LIN {X 0,Y 397.107,Z 581.021,A -85,B 0,C 180,E1 -11285.734,E2 -11285.734} C_VEL
LIN {X 0,Y 397.113,Z 581.016,A -85,B 0,C 180,E1 -11289.576,E2 -11289.576} C_VEL
LIN {X 0,Y 397.111,Z 581.016,A -85,B 0,C 180,E1 -11292.26,E2 -11292.26} C_VEL
LIN {X 0,Y 397.161,Z 581.009,A -85,B 0,C 180,E1 -11296.36,E2 -11296.36} C_VEL
LIN {X 0,Y 397.119,Z 581.014,A -85,B 0,C 180,E1 -11299.55,E2 -11299.55} C_VEL
LIN {X 0,Y 397.094,Z 581.019,A -85,B 0,C 180,E1 -11302.789,E2 -11302.789} C_VEL
LIN {X 0,Y 397.113,Z 581.011,A -85,B 0,C 180,E1 -11306.281,E2 -11306.281} C_VEL
LIN {X 0,Y 397.08,Z 581.018,A -85,B 0,C 180,E1 -11309.118,E2 -11309.118} C_VEL
LIN {X 0,Y 397.188,Z 581.007,A -85,B 0,C 180,E1 -11312.609,E2 -11312.609} C_VEL
LIN {X 0,Y 397.125,Z 581.014,A -85,B 0,C 180,E1 -11315.981,E2 -11315.981} C_VEL
LIN {X 0,Y 397.131,Z 581.012,A -85,B 0,C 180,E1 -11319.704,E2 -11319.704} C_VEL
LIN {X 0,Y 397.173,Z 581,A -85,B 0,C 180,E1 -11322.844,E2 -11322.844} C_VEL
LIN {X 0,Y 397.22,Z 581.007,A -85,B 0,C 180,E1 -11326.702,E2 -11326.702} C_VEL
LIN {X 0,Y 397.21,Z 580.998,A -85,B 0,C 180,E1 -11329.809,E2 -11329.809} C_VEL
LIN {X 0,Y 397.343,Z 580.986,A -85,B 0,C 180,E1 -11332.888,E2 -11332.888} C_VEL
LIN {X 0,Y 397.254,Z 581.001,A -85,B 0,C 180,E1 -11334.925,E2 -11334.925} C_VEL
LIN {X 0,Y 397.443,Z 580.964,A -85,B 0,C 180,E1 -11337.973,E2 -11337.973} C_VEL
LIN {X 0,Y 397.573,Z 580.952,A -85,B 0,C 180,E1 -11340,E2 -11340} C_VEL
LIN {X 0,Y 397.374,Z 580.984,A -85,B 0,C 180,E1 -11343.041,E2 -11343.041} C_VEL
LIN {X 0,Y 397.339,Z 580.977,A -85,B 0,C 180,E1 -11346.622,E2 -11346.622} C_VEL
LIN {X 0,Y 397.244,Z 581.002,A -85,B 0,C 180,E1 -11349.162,E2 -11349.162} C_VEL
LIN {X 0,Y 397.211,Z 580.994,A -85,B 0,C 180,E1 -11352.258,E2 -11352.258} C_VEL
LIN {X 0,Y 397.17,Z 581.011,A -85,B 0,C 180,E1 -11355.392,E2 -11355.392} C_VEL
LIN {X 0,Y 397.153,Z 581.004,A -85,B 0,C 180,E1 -11358.574,E2 -11358.574} C_VEL
LIN {X 0,Y 397.087,Z 581.019,A -85,B 0,C 180,E1 -11361.819,E2 -11361.819} C_VEL
LIN {X 0,Y 397.145,Z 581.011,A -85,B 0,C 180,E1 -11365.513,E2 -11365.513} C_VEL
LIN {X 0,Y 397.12,Z 581.016,A -85,B 0,C 180,E1 -11368.544,E2 -11368.544} C_VEL
LIN {X 0,Y 397.106,Z 581.017,A -85,B 0,C 180,E1 -11372.069,E2 -11372.069} C_VEL
LIN {X 0,Y 397.114,Z 581.019,A -85,B 0,C 180,E1 -11375.504,E2 -11375.504} C_VEL
LIN {X 0,Y 397.13,Z 581.017,A -85,B 0,C 180,E1 -11378.863,E2 -11378.863} C_VEL
LIN {X 0,Y 397.111,Z 580.995,A -85,B 0,C 180,E1 -11382.262,E2 -11382.262} C_VEL
LIN {X 0,Y 397.085,Z 581.023,A -85,B 0,C 180,E1 -11385.069,E2 -11385.069} C_VEL
LIN {X 0,Y 397.062,Z 581.012,A -85,B 0,C 180,E1 -11388.022,E2 -11388.022} C_VEL
LIN {X 0,Y 397.129,Z 581.012,A -85,B 0,C 180,E1 -11391.139,E2 -11391.139} C_VEL
LIN {X 0,Y 397.118,Z 581.016,A -85,B 0,C 180,E1 -11394.497,E2 -11394.497} C_VEL
LIN {X 0,Y 397.104,Z 581.02,A -85,B 0,C 180,E1 -11397.531,E2 -11397.531} C_VEL
LIN {X 0,Y 398.153,Z 583.972,A -85,B 0,C 180,E1 -11397.677,E2 -11397.677} C_VEL
LIN {X 0,Y 404.838,Z 599.166,A -85,B 0,C 180,E1 -11398.379,E2 -11398.379} C_VEL
LIN {X 0,Y 403.608,Z 681.671,A -85,B 0,C 180,E1 -11399.888,E2 -11399.888} C_VEL
LIN {X 0,Y 403.342,Z 694.362,A -85,B 0,C 180,E1 -11400.305,E2 -11400.305} C_VEL
LIN {X 0,Y 402.939,Z 705.504,A -85,B 0,C 180,E1 -11400.844,E2 -11400.844} C_VEL
LIN {X 0,Y 402.29,Z 716.836,A -85,B 0,C 180,E1 -11401.573,E2 -11401.573} C_VEL
LIN {X 0,Y 401.469,Z 728.036,A -85,B 0,C 180,E1 -11402.503,E2 -11402.503} C_VEL
LIN {X 0,Y 400.575,Z 738.584,A -85,B 0,C 180,E1 -11403.604,E2 -11403.604} C_VEL
LIN {X 0,Y 399.779,Z 747.58,A -85,B 0,C 180,E1 -11404.767,E2 -11404.767} C_VEL
LIN {X 0,Y 398.991,Z 755.975,A -85,B 0,C 180,E1 -11406.101,E2 -11406.101} C_VEL
LIN {X 0,Y 398.143,Z 764.097,A -85,B 0,C 180,E1 -11407.697,E2 -11407.697} C_VEL
LIN {X 0,Y 397.527,Z 770.543,A -85,B 0,C 180,E1 -11409.294,E2 -11409.294} C_VEL
LIN {X 0,Y 397.01,Z 775.554,A -85,B 0,C 180,E1 -11410.884,E2 -11410.884} C_VEL
LIN {X 0,Y 396.638,Z 779.358,A -85,B 0,C 180,E1 -11412.469,E2 -11412.469} C_VEL
LIN {X 0,Y 396.452,Z 781.287,A -85,B 0,C 180,E1 -11413.523,E2 -11413.523} C_VEL
LIN {X 0,Y 396.255,Z 782.789,A -85,B 0,C 180,E1 -11414.572,E2 -11414.572} C_VEL
LIN {X 0,Y 396.14,Z 783.814,A -85,B 0,C 180,E1 -11415.619,E2 -11415.619} C_VEL
LIN {X 0,Y 396.103,Z 784.664,A -85,B 0,C 180,E1 -11417.707,E2 -11417.707} C_VEL
LIN {X 0,Y 396.063,Z 784.463,A -85,B 0,C 180,E1 -11418.744,E2 -11418.744} C_VEL
LIN {X 0,Y 396.135,Z 782.858,A -85,B 0,C 180,E1 -11420.812,E2 -11420.812} C_VEL
LIN {X 0,Y 396.234,Z 781.448,A -85,B 0,C 180,E1 -11421.843,E2 -11421.843} C_VEL
LIN {X 0,Y 396.459,Z 779.154,A -85,B 0,C 180,E1 -11423.078,E2 -11423.078} C_VEL
LIN {X 0,Y 396.744,Z 774.546,A -85,B 0,C 180,E1 -11424.919,E2 -11424.919} C_VEL
LIN {X 0,Y 397.06,Z 769.443,A -85,B 0,C 180,E1 -11426.448,E2 -11426.448} C_VEL
LIN {X 0,Y 397.584,Z 763.023,A -85,B 0,C 180,E1 -11427.974,E2 -11427.974} C_VEL
LIN {X 0,Y 398.172,Z 755.074,A -85,B 0,C 180,E1 -11429.494,E2 -11429.494} C_VEL
LIN {X 0,Y 398.92,Z 746.903,A -85,B 0,C 180,E1 -11430.757,E2 -11430.757} C_VEL
LIN {X 0,Y 399.601,Z 736.901,A -85,B 0,C 180,E1 -11432.016,E2 -11432.016} C_VEL
LIN {X 0,Y 400.368,Z 725.703,A -85,B 0,C 180,E1 -11433.145,E2 -11433.145} C_VEL
LIN {X 0,Y 400.855,Z 718.327,A -85,B 0,C 180,E1 -11433.746,E2 -11433.746} C_VEL
LIN {X 0,Y 400.522,Z 713.137,A -85,B 0,C 180,E1 -11434.145,E2 -11434.145} C_VEL
LIN {X 0,Y 398.165,Z 704.558,A -85,B 0,C 180,E1 -11434.779,E2 -11434.779} C_VEL
LIN {X 0,Y 395.699,Z 695.737,A -85,B 0,C 180,E1 -11435.325,E2 -11435.325} C_VEL
LIN {X 0,Y 395.17,Z 690.125,A -85,B 0,C 180,E1 -11435.573,E2 -11435.573} C_VEL
LIN {X 0,Y 395.439,Z 677.057,A -85,B 0,C 180,E1 -11435.929,E2 -11435.929} C_VEL
LIN {X 0,Y 396.414,Z 599.082,A -85,B 0,C 180,E1 -11437.34,E2 -11437.34} C_VEL
LIN {X 0,Y 390.306,Z 581.87,A -85,B 0,C 180,E1 -11437.965,E2 -11437.965} C_VEL
LIN {X 0,Y 390.16,Z 581.883,A -85,B 0,C 180,E1 -11441.428,E2 -11441.428} C_VEL
LIN {X 0,Y 390.149,Z 581.885,A -85,B 0,C 180,E1 -11444.607,E2 -11444.607} C_VEL
LIN {X 0,Y 390.129,Z 581.891,A -85,B 0,C 180,E1 -11447.833,E2 -11447.833} C_VEL
LIN {X 0,Y 390.056,Z 581.893,A -85,B 0,C 180,E1 -11451.122,E2 -11451.122} C_VEL
LIN {X 0,Y 390.073,Z 581.895,A -85,B 0,C 180,E1 -11454.48,E2 -11454.48} C_VEL
LIN {X 0,Y 390.107,Z 581.919,A -85,B 0,C 180,E1 -11455.872,E2 -11455.872} C_VEL
LIN {X 0,Y 396.737,Z 599.495,A -85,B 0,C 180,E1 -11456.558,E2 -11456.558} C_VEL
LIN {X 0,Y 395.49,Z 682.574,A -85,B 0,C 180,E1 -11458.183,E2 -11458.183} C_VEL
LIN {X 0,Y 395.145,Z 696.043,A -85,B 0,C 180,E1 -11458.663,E2 -11458.663} C_VEL
LIN {X 0,Y 394.709,Z 707.466,A -85,B 0,C 180,E1 -11459.253,E2 -11459.253} C_VEL
LIN {X 0,Y 394.113,Z 718.824,A -85,B 0,C 180,E1 -11460.027,E2 -11460.027} C_VEL
LIN {X 0,Y 393.39,Z 730.372,A -85,B 0,C 180,E1 -11461.046,E2 -11461.046} C_VEL
LIN {X 0,Y 392.604,Z 740.657,A -85,B 0,C 180,E1 -11462.177,E2 -11462.177} C_VEL
LIN {X 0,Y 391.83,Z 750.29,A -85,B 0,C 180,E1 -11463.487,E2 -11463.487} C_VEL
LIN {X 0,Y 391.14,Z 758.584,A -85,B 0,C 180,E1 -11464.884,E2 -11464.884} C_VEL
LIN {X 0,Y 390.469,Z 766.071,A -85,B 0,C 180,E1 -11466.438,E2 -11466.438} C_VEL
LIN {X 0,Y 390.018,Z 772.477,A -85,B 0,C 180,E1 -11468.109,E2 -11468.109} C_VEL
LIN {X 0,Y 389.575,Z 777.532,A -85,B 0,C 180,E1 -11469.822,E2 -11469.822} C_VEL
LIN {X 0,Y 389.315,Z 780.786,A -85,B 0,C 180,E1 -11471.272,E2 -11471.272} C_VEL
LIN {X 0,Y 389.164,Z 782.437,A -85,B 0,C 180,E1 -11472.232,E2 -11472.232} C_VEL
LIN {X 0,Y 389.023,Z 784.323,A -85,B 0,C 180,E1 -11473.728,E2 -11473.728} C_VEL
LIN {X 0,Y 388.955,Z 785.325,A -85,B 0,C 180,E1 -11475.195,E2 -11475.195} C_VEL
LIN {X 0,Y 388.95,Z 785.526,A -85,B 0,C 180,E1 -11476.636,E2 -11476.636} C_VEL
LIN {X 0,Y 389.025,Z 784.989,A -85,B 0,C 180,E1 -11478.054,E2 -11478.054} C_VEL
LIN {X 0,Y 389.185,Z 783.734,A -85,B 0,C 180,E1 -11479.451,E2 -11479.451} C_VEL
LIN {X 0,Y 389.545,Z 780.384,A -85,B 0,C 180,E1 -11481.54,E2 -11481.54} C_VEL
LIN {X 0,Y 389.864,Z 776.967,A -85,B 0,C 180,E1 -11483.005,E2 -11483.005} C_VEL
LIN {X 0,Y 390.382,Z 771.36,A -85,B 0,C 180,E1 -11484.824,E2 -11484.824} C_VEL
LIN {X 0,Y 391.044,Z 764.821,A -85,B 0,C 180,E1 -11486.451,E2 -11486.451} C_VEL
LIN {X 0,Y 391.877,Z 756.375,A -85,B 0,C 180,E1 -11488.106,E2 -11488.106} C_VEL
LIN {X 0,Y 392.628,Z 748.547,A -85,B 0,C 180,E1 -11489.349,E2 -11489.349} C_VEL
LIN {X 0,Y 393.456,Z 739.523,A -85,B 0,C 180,E1 -11490.529,E2 -11490.529} C_VEL
LIN {X 0,Y 394.26,Z 728.785,A -85,B 0,C 180,E1 -11491.666,E2 -11491.666} C_VEL
LIN {X 0,Y 395.106,Z 716.39,A -85,B 0,C 180,E1 -11492.689,E2 -11492.689} C_VEL
LIN {X 0,Y 395.759,Z 704.167,A -85,B 0,C 180,E1 -11493.452,E2 -11493.452} C_VEL
LIN {X 0,Y 396.157,Z 690.604,A -85,B 0,C 180,E1 -11494.055,E2 -11494.055} C_VEL
LIN {X 0,Y 396.419,Z 678.086,A -85,B 0,C 180,E1 -11494.404,E2 -11494.404} C_VEL
LIN {X 0,Y 397.8,Z 600.33,A -85,B 0,C 180,E1 -11495.932,E2 -11495.932} C_VEL
LIN {X 0,Y 390.166,Z 582.414,A -85,B 0,C 180,E1 -11496.794,E2 -11496.794} C_VEL
LIN {X 0,Y 390.076,Z 581.896,A -85,B 0,C 180,E1 -11496.817,E2 -11496.817} C_VEL
LIN {X 0,Y 390.096,Z 581.894,A -85,B 0,C 180,E1 -11499.983,E2 -11499.983} C_VEL
LIN {X 0,Y 390.13,Z 581.889,A -85,B 0,C 180,E1 -11503.248,E2 -11503.248} C_VEL
LIN {X 0,Y 390.186,Z 581.883,A -85,B 0,C 180,E1 -11506.561,E2 -11506.561} C_VEL
LIN {X 0,Y 390.171,Z 581.883,A -85,B 0,C 180,E1 -11509.623,E2 -11509.623} C_VEL
LIN {X 0,Y 390.31,Z 581.866,A -85,B 0,C 180,E1 -11512.759,E2 -11512.759} C_VEL
LIN {X 0,Y 390.225,Z 581.875,A -85,B 0,C 180,E1 -11514.833,E2 -11514.833} C_VEL
LIN {X 0,Y 390.412,Z 581.849,A -85,B 0,C 180,E1 -11517.937,E2 -11517.937} C_VEL
LIN {X 0,Y 390.543,Z 581.837,A -85,B 0,C 180,E1 -11520,E2 -11520} C_VEL
LIN {X 0,Y 390.308,Z 581.861,A -85,B 0,C 180,E1 -11523.097,E2 -11523.097} C_VEL
LIN {X 0,Y 390.33,Z 581.863,A -85,B 0,C 180,E1 -11526.202,E2 -11526.202} C_VEL
LIN {X 0,Y 390.201,Z 581.873,A -85,B 0,C 180,E1 -11529.329,E2 -11529.329} C_VEL
LIN {X 0,Y 390.169,Z 581.88,A -85,B 0,C 180,E1 -11532.483,E2 -11532.483} C_VEL
LIN {X 0,Y 390.131,Z 581.882,A -85,B 0,C 180,E1 -11535.677,E2 -11535.677} C_VEL
LIN {X 0,Y 390.097,Z 581.888,A -85,B 0,C 180,E1 -11538.923,E2 -11538.923} C_VEL
LIN {X 0,Y 390.033,Z 581.899,A -85,B 0,C 180,E1 -11542.235,E2 -11542.235} C_VEL
LIN {X 0,Y 390.112,Z 581.889,A -85,B 0,C 180,E1 -11545.744,E2 -11545.744} C_VEL
LIN {X 0,Y 390.059,Z 581.896,A -85,B 0,C 180,E1 -11549.11,E2 -11549.11} C_VEL
LIN {X 0,Y 390.037,Z 581.899,A -85,B 0,C 180,E1 -11552.722,E2 -11552.722} C_VEL
LIN {X 0,Y 390.052,Z 581.897,A -85,B 0,C 180,E1 -11555.826,E2 -11555.826} C_VEL
LIN {X 0,Y 390.07,Z 581.893,A -85,B 0,C 180,E1 -11559.22,E2 -11559.22} C_VEL
LIN {X 0,Y 390.116,Z 581.891,A -85,B 0,C 180,E1 -11562.388,E2 -11562.388} C_VEL
LIN {X 0,Y 390.057,Z 581.897,A -85,B 0,C 180,E1 -11565.358,E2 -11565.358} C_VEL
LIN {X 0,Y 390.065,Z 581.898,A -85,B 0,C 180,E1 -11568.192,E2 -11568.192} C_VEL
LIN {X 0,Y 390.092,Z 581.894,A -85,B 0,C 180,E1 -11570.909,E2 -11570.909} C_VEL
LIN {X 0,Y 390.084,Z 581.894,A -85,B 0,C 180,E1 -11574.794,E2 -11574.794} C_VEL
LIN {X 0,Y 390.073,Z 582.026,A -85,B 0,C 180,E1 -11578.363,E2 -11578.363} C_VEL
LIN {X 0,Y 392.97,Z 594.47,A -85,B 0,C 180,E1 -11581.127,E2 -11581.127} C_VEL
LIN {X 0,Y 394.598,Z 603.068,A -85,B 0,C 180,E1 -11582.94,E2 -11582.94} C_VEL
LIN {X 0,Y 393.842,Z 613.598,A -85,B 0,C 180,E1 -11584.925,E2 -11584.925} C_VEL
LIN {X 0,Y 392.147,Z 635.612,A -85,B 0,C 180,E1 -11588.996,E2 -11588.996} C_VEL
LIN {X 0,Y 392.035,Z 636.9,A -85,B 0,C 180,E1 -11589.231,E2 -11589.231} C_VEL
LIN {X 0,Y 395.926,Z 664.717,A -85,B 0,C 180,E1 -11590.051,E2 -11590.051} C_VEL
LIN {X 0,Y 396.965,Z 675.261,A -85,B 0,C 180,E1 -11590.325,E2 -11590.325} C_VEL
LIN {X 0,Y 395.717,Z 747.647,A -85,B 0,C 180,E1 -11591.759,E2 -11591.759} C_VEL
LIN {X 0,Y 395.033,Z 761.284,A -85,B 0,C 180,E1 -11592.229,E2 -11592.229} C_VEL
LIN {X 0,Y 394.133,Z 774.25,A -85,B 0,C 180,E1 -11592.89,E2 -11592.89} C_VEL
LIN {X 0,Y 393.186,Z 786.925,A -85,B 0,C 180,E1 -11593.783,E2 -11593.783} C_VEL
LIN {X 0,Y 392.18,Z 798.275,A -85,B 0,C 180,E1 -11594.807,E2 -11594.807} C_VEL
LIN {X 0,Y 391.42,Z 808.805,A -85,B 0,C 180,E1 -11596.003,E2 -11596.003} C_VEL
LIN {X 0,Y 390.496,Z 817.885,A -85,B 0,C 180,E1 -11597.264,E2 -11597.264} C_VEL
LIN {X 0,Y 389.799,Z 827.014,A -85,B 0,C 180,E1 -11598.824,E2 -11598.824} C_VEL
LIN {X 0,Y 389.327,Z 834.372,A -85,B 0,C 180,E1 -11600.388,E2 -11600.388} C_VEL
LIN {X 0,Y 389.037,Z 841.107,A -85,B 0,C 180,E1 -11602.213,E2 -11602.213} C_VEL
LIN {X 0,Y 388.903,Z 845.58,A -85,B 0,C 180,E1 -11603.775,E2 -11603.775} C_VEL
LIN {X 0,Y 388.942,Z 847.974,A -85,B 0,C 180,E1 -11604.817,E2 -11604.817} C_VEL
LIN {X 0,Y 388.856,Z 849.875,A -85,B 0,C 180,E1 -11605.854,E2 -11605.854} C_VEL
LIN {X 0,Y 388.997,Z 851.337,A -85,B 0,C 180,E1 -11606.893,E2 -11606.893} C_VEL
LIN {X 0,Y 389.023,Z 852.379,A -85,B 0,C 180,E1 -11607.929,E2 -11607.929} C_VEL
LIN {X 0,Y 389.002,Z 853.016,A -85,B 0,C 180,E1 -11608.965,E2 -11608.965} C_VEL
LIN {X 0,Y 388.967,Z 853.206,A -85,B 0,C 180,E1 -11610,E2 -11610} C_VEL
LIN {X 0,Y 389.002,Z 852.98,A -85,B 0,C 180,E1 -11611.035,E2 -11611.035} C_VEL
LIN {X 0,Y 389.049,Z 852.354,A -85,B 0,C 180,E1 -11612.07,E2 -11612.07} C_VEL
LIN {X 0,Y 389,Z 851.311,A -85,B 0,C 180,E1 -11613.107,E2 -11613.107} C_VEL
LIN {X 0,Y 388.869,Z 849.793,A -85,B 0,C 180,E1 -11614.146,E2 -11614.146} C_VEL
LIN {X 0,Y 388.926,Z 846.715,A -85,B 0,C 180,E1 -11615.704,E2 -11615.704} C_VEL
LIN {X 0,Y 388.935,Z 842.53,A -85,B 0,C 180,E1 -11617.267,E2 -11617.267} C_VEL
LIN {X 0,Y 389.207,Z 836.12,A -85,B 0,C 180,E1 -11619.091,E2 -11619.091} C_VEL
LIN {X 0,Y 389.596,Z 829.127,A -85,B 0,C 180,E1 -11620.655,E2 -11620.655} C_VEL
LIN {X 0,Y 390.39,Z 819.171,A -85,B 0,C 180,E1 -11622.476,E2 -11622.476} C_VEL
LIN {X 0,Y 391.218,Z 809.61,A -85,B 0,C 180,E1 -11623.878,E2 -11623.878} C_VEL
LIN {X 0,Y 392.057,Z 799.634,A -85,B 0,C 180,E1 -11625.065,E2 -11625.065} C_VEL
LIN {X 0,Y 393.058,Z 788.861,A -85,B 0,C 180,E1 -11626.089,E2 -11626.089} C_VEL
LIN {X 0,Y 394.062,Z 776.778,A -85,B 0,C 180,E1 -11626.98,E2 -11626.98} C_VEL
LIN {X 0,Y 394.884,Z 764.155,A -85,B 0,C 180,E1 -11627.678,E2 -11627.678} C_VEL
LIN {X 0,Y 395.592,Z 751.57,A -85,B 0,C 180,E1 -11628.147,E2 -11628.147} C_VEL
LIN {X 0,Y 395.948,Z 735.695,A -85,B 0,C 180,E1 -11628.498,E2 -11628.498} C_VEL
LIN {X 0,Y 396.808,Z 671.548,A -85,B 0,C 180,E1 -11629.684,E2 -11629.684} C_VEL
LIN {X 0,Y 392.936,Z 639.109,A -85,B 0,C 180,E1 -11630.548,E2 -11630.548} C_VEL
LIN {X 0,Y 392.608,Z 636.373,A -85,B 0,C 180,E1 -11630.635,E2 -11630.635} C_VEL
LIN {X 0,Y 394.524,Z 610.695,A -85,B 0,C 180,E1 -11634.7,E2 -11634.7} C_VEL
LIN {X 0,Y 394.953,Z 603.562,A -85,B 0,C 180,E1 -11635.846,E2 -11635.846} C_VEL
LIN {X 0,Y 391.748,Z 588.885,A -85,B 0,C 180,E1 -11638.47,E2 -11638.47} C_VEL
LIN {X 0,Y 390.068,Z 581.896,A -85,B 0,C 180,E1 -11639.78,E2 -11639.78} C_VEL
LIN {X 0,Y 390.042,Z 581.899,A -85,B 0,C 180,E1 -11642.721,E2 -11642.721} C_VEL
LIN {X 0,Y 390.056,Z 581.901,A -85,B 0,C 180,E1 -11645.825,E2 -11645.825} C_VEL
LIN {X 0,Y 390.071,Z 581.892,A -85,B 0,C 180,E1 -11649.218,E2 -11649.218} C_VEL
LIN {X 0,Y 390.077,Z 581.892,A -85,B 0,C 180,E1 -11652.379,E2 -11652.379} C_VEL
LIN {X 0,Y 390.101,Z 581.887,A -85,B 0,C 180,E1 -11656.105,E2 -11656.105} C_VEL
LIN {X 0,Y 390.078,Z 581.89,A -85,B 0,C 180,E1 -11659.173,E2 -11659.173} C_VEL
LIN {X 0,Y 390.042,Z 581.901,A -85,B 0,C 180,E1 -11662.448,E2 -11662.448} C_VEL
LIN {X 0,Y 390.062,Z 581.887,A -85,B 0,C 180,E1 -11666.044,E2 -11666.044} C_VEL
LIN {X 0,Y 390.042,Z 581.9,A -85,B 0,C 180,E1 -11668.497,E2 -11668.497} C_VEL
LIN {X 0,Y 390.11,Z 581.88,A -85,B 0,C 180,E1 -11672.069,E2 -11672.069} C_VEL
LIN {X 0,Y 390.072,Z 581.891,A -85,B 0,C 180,E1 -11675.519,E2 -11675.519} C_VEL
LIN {X 0,Y 390.047,Z 581.896,A -85,B 0,C 180,E1 -11678.877,E2 -11678.877} C_VEL
LIN {X 0,Y 390.12,Z 581.889,A -85,B 0,C 180,E1 -11682.166,E2 -11682.166} C_VEL
LIN {X 0,Y 390.135,Z 581.879,A -85,B 0,C 180,E1 -11685.392,E2 -11685.392} C_VEL
LIN {X 0,Y 390.14,Z 581.886,A -85,B 0,C 180,E1 -11688.571,E2 -11688.571} C_VEL
LIN {X 0,Y 390.298,Z 581.852,A -85,B 0,C 180,E1 -11692.032,E2 -11692.032} C_VEL
LIN {X 0,Y 390.226,Z 581.878,A -85,B 0,C 180,E1 -11694.833,E2 -11694.833} C_VEL
LIN {X 0,Y 390.412,Z 581.839,A -85,B 0,C 180,E1 -11697.937,E2 -11697.937} C_VEL
LIN {X 0,Y 390.543,Z 581.827,A -85,B 0,C 180,E1 -11700,E2 -11700} C_VEL
LIN {X 0,Y 390.308,Z 581.863,A -85,B 0,C 180,E1 -11703.097,E2 -11703.097} C_VEL
LIN {X 0,Y 390.295,Z 581.854,A -85,B 0,C 180,E1 -11706.616,E2 -11706.616} C_VEL
LIN {X 0,Y 390.196,Z 581.879,A -85,B 0,C 180,E1 -11709.329,E2 -11709.329} C_VEL
LIN {X 0,Y 390.186,Z 581.875,A -85,B 0,C 180,E1 -11713.439,E2 -11713.439} C_VEL
LIN {X 0,Y 390.14,Z 581.881,A -85,B 0,C 180,E1 -11717.308,E2 -11717.308} C_VEL
LIN {X 0,Y 390.079,Z 581.888,A -85,B 0,C 180,E1 -11720.47,E2 -11720.47} C_VEL
LIN {X 0,Y 390.07,Z 581.887,A -85,B 0,C 180,E1 -11724.481,E2 -11724.481} C_VEL
LIN {X 0,Y 390.109,Z 581.888,A -85,B 0,C 180,E1 -11728.026,E2 -11728.026} C_VEL
LIN {X 0,Y 390.043,Z 581.9,A -85,B 0,C 180,E1 -11731.503,E2 -11731.503} C_VEL
LIN {X 0,Y 390.08,Z 581.891,A -85,B 0,C 180,E1 -11735.208,E2 -11735.208} C_VEL
LIN {X 0,Y 390.089,Z 581.897,A -85,B 0,C 180,E1 -11739.093,E2 -11739.093} C_VEL
LIN {X 0,Y 390.077,Z 581.87,A -85,B 0,C 180,E1 -11742.381,E2 -11742.381} C_VEL
LIN {X 0,Y 390.051,Z 581.894,A -85,B 0,C 180,E1 -11746.115,E2 -11746.115} C_VEL
LIN {X 0,Y 390.053,Z 581.899,A -85,B 0,C 180,E1 -11749.561,E2 -11749.561} C_VEL
LIN {X 0,Y 390.043,Z 581.89,A -85,B 0,C 180,E1 -11752.45,E2 -11752.45} C_VEL
LIN {X 0,Y 390.066,Z 581.896,A -85,B 0,C 180,E1 -11755.976,E2 -11755.976} C_VEL
LIN {X 0,Y 390.061,Z 581.897,A -85,B 0,C 180,E1 -11757.098,E2 -11757.098} C_VEL
LIN {X 0,Y 391.138,Z 584.861,A -85,B 0,C 180,E1 -11757.24,E2 -11757.24} C_VEL
LIN {X 0,Y 398.258,Z 600.928,A -85,B 0,C 180,E1 -11758.011,E2 -11758.011} C_VEL
LIN {X 0,Y 397.013,Z 682.018,A -85,B 0,C 180,E1 -11759.518,E2 -11759.518} C_VEL
LIN {X 0,Y 396.752,Z 694.64,A -85,B 0,C 180,E1 -11759.937,E2 -11759.937} C_VEL
LIN {X 0,Y 396.302,Z 705.838,A -85,B 0,C 180,E1 -11760.48,E2 -11760.48} C_VEL
LIN {X 0,Y 395.646,Z 717.052,A -85,B 0,C 180,E1 -11761.205,E2 -11761.205} C_VEL
LIN {X 0,Y 394.79,Z 728.228,A -85,B 0,C 180,E1 -11762.142,E2 -11762.142} C_VEL
LIN {X 0,Y 393.825,Z 739.065,A -85,B 0,C 180,E1 -11763.286,E2 -11763.286} C_VEL
LIN {X 0,Y 392.902,Z 748.814,A -85,B 0,C 180,E1 -11764.578,E2 -11764.578} C_VEL
LIN {X 0,Y 391.946,Z 758.19,A -85,B 0,C 180,E1 -11766.133,E2 -11766.133} C_VEL
LIN {X 0,Y 391.205,Z 765.125,A -85,B 0,C 180,E1 -11767.558,E2 -11767.558} C_VEL
LIN {X 0,Y 390.645,Z 770.502,A -85,B 0,C 180,E1 -11768.912,E2 -11768.912} C_VEL
LIN {X 0,Y 390.075,Z 775.688,A -85,B 0,C 180,E1 -11770.53,E2 -11770.53} C_VEL
LIN {X 0,Y 389.647,Z 779.619,A -85,B 0,C 180,E1 -11772.144,E2 -11772.144} C_VEL
LIN {X 0,Y 389.458,Z 781.604,A -85,B 0,C 180,E1 -11773.219,E2 -11773.219} C_VEL
LIN {X 0,Y 389.245,Z 783.166,A -85,B 0,C 180,E1 -11774.287,E2 -11774.287} C_VEL
LIN {X 0,Y 389.094,Z 784.294,A -85,B 0,C 180,E1 -11775.353,E2 -11775.353} C_VEL
LIN {X 0,Y 389.053,Z 785.244,A -85,B 0,C 180,E1 -11777.481,E2 -11777.481} C_VEL
LIN {X 0,Y 389.007,Z 785.138,A -85,B 0,C 180,E1 -11778.537,E2 -11778.537} C_VEL
LIN {X 0,Y 389.067,Z 783.643,A -85,B 0,C 180,E1 -11780.644,E2 -11780.644} C_VEL
LIN {X 0,Y 389.148,Z 782.309,A -85,B 0,C 180,E1 -11781.693,E2 -11781.693} C_VEL
LIN {X 0,Y 389.382,Z 779.851,A -85,B 0,C 180,E1 -11783.075,E2 -11783.075} C_VEL
LIN {X 0,Y 389.676,Z 775.632,A -85,B 0,C 180,E1 -11784.826,E2 -11784.826} C_VEL
LIN {X 0,Y 389.997,Z 770.674,A -85,B 0,C 180,E1 -11786.384,E2 -11786.384} C_VEL
LIN {X 0,Y 390.525,Z 764.398,A -85,B 0,C 180,E1 -11787.937,E2 -11787.937} C_VEL
LIN {X 0,Y 391.1,Z 756.611,A -85,B 0,C 180,E1 -11789.485,E2 -11789.485} C_VEL
LIN {X 0,Y 391.854,Z 748.635,A -85,B 0,C 180,E1 -11790.771,E2 -11790.771} C_VEL
LIN {X 0,Y 392.595,Z 738.95,A -85,B 0,C 180,E1 -11792.052,E2 -11792.052} C_VEL
LIN {X 0,Y 393.34,Z 728.066,A -85,B 0,C 180,E1 -11793.201,E2 -11793.201} C_VEL
LIN {X 0,Y 394.063,Z 717.452,A -85,B 0,C 180,E1 -11794.091,E2 -11794.091} C_VEL
LIN {X 0,Y 394.692,Z 704.664,A -85,B 0,C 180,E1 -11794.916,E2 -11794.916} C_VEL
LIN {X 0,Y 395.13,Z 691.574,A -85,B 0,C 180,E1 -11795.518,E2 -11795.518} C_VEL
LIN {X 0,Y 395.17,Z 690.125,A -85,B 0,C 180,E1 -11795.573,E2 -11795.573} C_VEL
LIN {X 0,Y 394.652,Z 684.425,A -85,B 0,C 180,E1 -11795.786,E2 -11795.786} C_VEL
LIN {X 0,Y 389.395,Z 665.772,A -85,B 0,C 180,E1 -11796.397,E2 -11796.397} C_VEL
LIN {X 0,Y 388.838,Z 659.957,A -85,B 0,C 180,E1 -11796.524,E2 -11796.524} C_VEL
LIN {X 0,Y 389.489,Z 600.174,A -85,B 0,C 180,E1 -11797.63,E2 -11797.63} C_VEL
LIN {X 0,Y 383.259,Z 582.747,A -85,B 0,C 180,E1 -11798.27,E2 -11798.27} C_VEL
LIN {X 0,Y 383.109,Z 582.763,A -85,B 0,C 180,E1 -11801.641,E2 -11801.641} C_VEL
LIN {X 0,Y 383.114,Z 582.76,A -85,B 0,C 180,E1 -11804.881,E2 -11804.881} C_VEL
LIN {X 0,Y 383.091,Z 582.768,A -85,B 0,C 180,E1 -11808.172,E2 -11808.172} C_VEL
LIN {X 0,Y 382.993,Z 582.775,A -85,B 0,C 180,E1 -11811.53,E2 -11811.53} C_VEL
LIN {X 0,Y 383.056,Z 582.768,A -85,B 0,C 180,E1 -11815.25,E2 -11815.25} C_VEL
LIN {X 0,Y 383.057,Z 582.769,A -85,B 0,C 180,E1 -11815.504,E2 -11815.504} C_VEL
LIN {X 0,Y 387.907,Z 595.517,A -85,B 0,C 180,E1 -11816.041,E2 -11816.041} C_VEL
LIN {X 0,Y 390.045,Z 601.164,A -85,B 0,C 180,E1 -11816.265,E2 -11816.265} C_VEL
LIN {X 0,Y 388.688,Z 683.075,A -85,B 0,C 180,E1 -11817.894,E2 -11817.894} C_VEL
LIN {X 0,Y 388.347,Z 696.518,A -85,B 0,C 180,E1 -11818.38,E2 -11818.38} C_VEL
LIN {X 0,Y 387.784,Z 709.508,A -85,B 0,C 180,E1 -11819.073,E2 -11819.073} C_VEL
LIN {X 0,Y 387.095,Z 721.91,A -85,B 0,C 180,E1 -11819.979,E2 -11819.979} C_VEL
LIN {X 0,Y 386.313,Z 733.533,A -85,B 0,C 180,E1 -11821.07,E2 -11821.07} C_VEL
LIN {X 0,Y 385.548,Z 743.292,A -85,B 0,C 180,E1 -11822.22,E2 -11822.22} C_VEL
LIN {X 0,Y 384.746,Z 752.441,A -85,B 0,C 180,E1 -11823.542,E2 -11823.542} C_VEL
LIN {X 0,Y 384.093,Z 760.013,A -85,B 0,C 180,E1 -11824.874,E2 -11824.874} C_VEL
LIN {X 0,Y 383.478,Z 766.506,A -85,B 0,C 180,E1 -11826.255,E2 -11826.255} C_VEL
LIN {X 0,Y 383.035,Z 772.783,A -85,B 0,C 180,E1 -11827.91,E2 -11827.91} C_VEL
LIN {X 0,Y 382.578,Z 777.551,A -85,B 0,C 180,E1 -11829.507,E2 -11829.507} C_VEL
LIN {X 0,Y 382.22,Z 781.806,A -85,B 0,C 180,E1 -11831.447,E2 -11831.447} C_VEL
LIN {X 0,Y 382.011,Z 784.041,A -85,B 0,C 180,E1 -11832.897,E2 -11832.897} C_VEL
LIN {X 0,Y 381.904,Z 785.475,A -85,B 0,C 180,E1 -11834.369,E2 -11834.369} C_VEL
LIN {X 0,Y 381.876,Z 786.127,A -85,B 0,C 180,E1 -11835.868,E2 -11835.868} C_VEL
LIN {X 0,Y 381.936,Z 785.973,A -85,B 0,C 180,E1 -11837.393,E2 -11837.393} C_VEL
LIN {X 0,Y 382.043,Z 784.957,A -85,B 0,C 180,E1 -11838.956,E2 -11838.956} C_VEL
LIN {X 0,Y 382.287,Z 783.003,A -85,B 0,C 180,E1 -11840.544,E2 -11840.544} C_VEL
LIN {X 0,Y 382.654,Z 780.005,A -85,B 0,C 180,E1 -11842.161,E2 -11842.161} C_VEL
LIN {X 0,Y 383.11,Z 775.103,A -85,B 0,C 180,E1 -11844.054,E2 -11844.054} C_VEL
LIN {X 0,Y 383.726,Z 769.014,A -85,B 0,C 180,E1 -11845.825,E2 -11845.825} C_VEL
LIN {X 0,Y 384.423,Z 762.843,A -85,B 0,C 180,E1 -11847.24,E2 -11847.24} C_VEL
LIN {X 0,Y 385.329,Z 754.263,A -85,B 0,C 180,E1 -11848.824,E2 -11848.824} C_VEL
LIN {X 0,Y 386.27,Z 744.463,A -85,B 0,C 180,E1 -11850.277,E2 -11850.277} C_VEL
LIN {X 0,Y 387.116,Z 735.148,A -85,B 0,C 180,E1 -11851.391,E2 -11851.391} C_VEL
LIN {X 0,Y 387.925,Z 724.557,A -85,B 0,C 180,E1 -11852.413,E2 -11852.413} C_VEL
LIN {X 0,Y 388.691,Z 712.241,A -85,B 0,C 180,E1 -11853.343,E2 -11853.343} C_VEL
LIN {X 0,Y 389.318,Z 699.489,A -85,B 0,C 180,E1 -11854.057,E2 -11854.057} C_VEL
LIN {X 0,Y 389.64,Z 686.186,A -85,B 0,C 180,E1 -11854.567,E2 -11854.567} C_VEL
LIN {X 0,Y 390.131,Z 660.878,A -85,B 0,C 180,E1 -11855.112,E2 -11855.112} C_VEL
LIN {X 0,Y 391.319,Z 602.375,A -85,B 0,C 180,E1 -11856.289,E2 -11856.289} C_VEL
LIN {X 0,Y 384.084,Z 585.668,A -85,B 0,C 180,E1 -11857.126,E2 -11857.126} C_VEL
LIN {X 0,Y 383.022,Z 582.777,A -85,B 0,C 180,E1 -11857.29,E2 -11857.29} C_VEL
LIN {X 0,Y 383.052,Z 582.772,A -85,B 0,C 180,E1 -11860.716,E2 -11860.716} C_VEL
LIN {X 0,Y 383.073,Z 582.769,A -85,B 0,C 180,E1 -11864.026,E2 -11864.026} C_VEL
LIN {X 0,Y 383.134,Z 582.76,A -85,B 0,C 180,E1 -11867.284,E2 -11867.284} C_VEL
LIN {X 0,Y 383.148,Z 582.758,A -85,B 0,C 180,E1 -11870.498,E2 -11870.498} C_VEL
LIN {X 0,Y 383.265,Z 582.744,A -85,B 0,C 180,E1 -11872.625,E2 -11872.625} C_VEL
LIN {X 0,Y 383.197,Z 582.751,A -85,B 0,C 180,E1 -11874.738,E2 -11874.738} C_VEL
LIN {X 0,Y 383.379,Z 582.725,A -85,B 0,C 180,E1 -11877.899,E2 -11877.899} C_VEL
LIN {X 0,Y 383.512,Z 582.713,A -85,B 0,C 180,E1 -11880,E2 -11880} C_VEL
LIN {X 0,Y 383.245,Z 582.74,A -85,B 0,C 180,E1 -11883.154,E2 -11883.154} C_VEL
LIN {X 0,Y 383.285,Z 582.739,A -85,B 0,C 180,E1 -11886.316,E2 -11886.316} C_VEL
LIN {X 0,Y 383.148,Z 582.752,A -85,B 0,C 180,E1 -11889.502,E2 -11889.502} C_VEL
LIN {X 0,Y 383.133,Z 582.753,A -85,B 0,C 180,E1 -11892.716,E2 -11892.716} C_VEL
LIN {X 0,Y 383.073,Z 582.762,A -85,B 0,C 180,E1 -11895.974,E2 -11895.974} C_VEL
LIN {X 0,Y 383.052,Z 582.764,A -85,B 0,C 180,E1 -11899.284,E2 -11899.284} C_VEL
LIN {X 0,Y 383.03,Z 582.766,A -85,B 0,C 180,E1 -11903.451,E2 -11903.451} C_VEL
LIN {X 0,Y 383.073,Z 582.768,A -85,B 0,C 180,E1 -11906.124,E2 -11906.124} C_VEL
LIN {X 0,Y 383.043,Z 582.771,A -85,B 0,C 180,E1 -11908.493,E2 -11908.493} C_VEL
LIN {X 0,Y 383,Z 582.78,A -85,B 0,C 180,E1 -11912.427,E2 -11912.427} C_VEL
LIN {X 0,Y 383.021,Z 582.774,A -85,B 0,C 180,E1 -11915.956,E2 -11915.956} C_VEL
LIN {X 0,Y 383.018,Z 582.771,A -85,B 0,C 180,E1 -11919.589,E2 -11919.589} C_VEL
LIN {X 0,Y 383.061,Z 582.771,A -85,B 0,C 180,E1 -11922.789,E2 -11922.789} C_VEL
LIN {X 0,Y 383.004,Z 582.776,A -85,B 0,C 180,E1 -11925.792,E2 -11925.792} C_VEL
LIN {X 0,Y 383.013,Z 582.777,A -85,B 0,C 180,E1 -11928.792,E2 -11928.792} C_VEL
LIN {X 0,Y 383.001,Z 582.779,A -85,B 0,C 180,E1 -11932.096,E2 -11932.096} C_VEL
LIN {X 0,Y 383.016,Z 582.773,A -85,B 0,C 180,E1 -11935.333,E2 -11935.333} C_VEL
LIN {X 0,Y 382.997,Z 582.806,A -85,B 0,C 180,E1 -11937.928,E2 -11937.928} C_VEL
LIN {X 0,Y 385.695,Z 594.12,A -85,B 0,C 180,E1 -11940.53,E2 -11940.53} C_VEL
LIN {X 0,Y 387.675,Z 603.972,A -85,B 0,C 180,E1 -11942.661,E2 -11942.661} C_VEL
LIN {X 0,Y 387.405,Z 610.291,A -85,B 0,C 180,E1 -11943.902,E2 -11943.902} C_VEL
LIN {X 0,Y 385.455,Z 632.241,A -85,B 0,C 180,E1 -11948.052,E2 -11948.052} C_VEL
LIN {X 0,Y 385.202,Z 636.244,A -85,B 0,C 180,E1 -11948.804,E2 -11948.804} C_VEL
LIN {X 0,Y 389.467,Z 666.747,A -85,B 0,C 180,E1 -11949.726,E2 -11949.726} C_VEL
LIN {X 0,Y 390.292,Z 677.193,A -85,B 0,C 180,E1 -11949.994,E2 -11949.994} C_VEL
LIN {X 0,Y 389.058,Z 746.85,A -85,B 0,C 180,E1 -11951.401,E2 -11951.401} C_VEL
LIN {X 0,Y 388.326,Z 760.514,A -85,B 0,C 180,E1 -11951.877,E2 -11951.877} C_VEL
LIN {X 0,Y 387.429,Z 772.979,A -85,B 0,C 180,E1 -11952.516,E2 -11952.516} C_VEL
LIN {X 0,Y 386.491,Z 785.003,A -85,B 0,C 180,E1 -11953.358,E2 -11953.358} C_VEL
LIN {X 0,Y 385.43,Z 796.582,A -85,B 0,C 180,E1 -11954.398,E2 -11954.398} C_VEL
LIN {X 0,Y 384.497,Z 807.558,A -85,B 0,C 180,E1 -11955.641,E2 -11955.641} C_VEL
LIN {X 0,Y 383.746,Z 815.701,A -85,B 0,C 180,E1 -11956.766,E2 -11956.766} C_VEL
LIN {X 0,Y 382.902,Z 825.076,A -85,B 0,C 180,E1 -11958.352,E2 -11958.352} C_VEL
LIN {X 0,Y 382.341,Z 832.675,A -85,B 0,C 180,E1 -11959.943,E2 -11959.943} C_VEL
LIN {X 0,Y 382.026,Z 838.804,A -85,B 0,C 180,E1 -11961.537,E2 -11961.537} C_VEL
LIN {X 0,Y 381.896,Z 843.664,A -85,B 0,C 180,E1 -11963.13,E2 -11963.13} C_VEL
LIN {X 0,Y 381.849,Z 847.388,A -85,B 0,C 180,E1 -11964.72,E2 -11964.72} C_VEL
LIN {X 0,Y 381.778,Z 849.278,A -85,B 0,C 180,E1 -11965.777,E2 -11965.777} C_VEL
LIN {X 0,Y 381.91,Z 850.734,A -85,B 0,C 180,E1 -11966.835,E2 -11966.835} C_VEL
LIN {X 0,Y 381.948,Z 851.775,A -85,B 0,C 180,E1 -11967.891,E2 -11967.891} C_VEL
LIN {X 0,Y 381.952,Z 852.406,A -85,B 0,C 180,E1 -11968.946,E2 -11968.946} C_VEL
LIN {X 0,Y 381.916,Z 852.582,A -85,B 0,C 180,E1 -11970,E2 -11970} C_VEL
LIN {X 0,Y 381.953,Z 852.35,A -85,B 0,C 180,E1 -11971.054,E2 -11971.054} C_VEL
LIN {X 0,Y 381.972,Z 851.713,A -85,B 0,C 180,E1 -11972.109,E2 -11972.109} C_VEL
LIN {X 0,Y 381.933,Z 850.661,A -85,B 0,C 180,E1 -11973.164,E2 -11973.164} C_VEL
LIN {X 0,Y 381.789,Z 849.125,A -85,B 0,C 180,E1 -11974.223,E2 -11974.223} C_VEL
LIN {X 0,Y 381.832,Z 845.608,A -85,B 0,C 180,E1 -11975.984,E2 -11975.984} C_VEL
LIN {X 0,Y 381.937,Z 840.169,A -85,B 0,C 180,E1 -11977.932,E2 -11977.932} C_VEL
LIN {X 0,Y 382.27,Z 833.197,A -85,B 0,C 180,E1 -11979.791,E2 -11979.791} C_VEL
LIN {X 0,Y 382.818,Z 826.057,A -85,B 0,C 180,E1 -11981.382,E2 -11981.382} C_VEL
LIN {X 0,Y 383.541,Z 817.237,A -85,B 0,C 180,E1 -11982.971,E2 -11982.971} C_VEL
LIN {X 0,Y 384.405,Z 807.529,A -85,B 0,C 180,E1 -11984.384,E2 -11984.384} C_VEL
LIN {X 0,Y 385.456,Z 797.029,A -85,B 0,C 180,E1 -11985.601,E2 -11985.601} C_VEL
LIN {X 0,Y 386.553,Z 785.724,A -85,B 0,C 180,E1 -11986.639,E2 -11986.639} C_VEL
LIN {X 0,Y 387.453,Z 773.992,A -85,B 0,C 180,E1 -11987.483,E2 -11987.483} C_VEL
LIN {X 0,Y 388.421,Z 761.057,A -85,B 0,C 180,E1 -11988.152,E2 -11988.152} C_VEL
LIN {X 0,Y 389.096,Z 748.328,A -85,B 0,C 180,E1 -11988.597,E2 -11988.597} C_VEL
LIN {X 0,Y 389.822,Z 701.665,A -85,B 0,C 180,E1 -11989.508,E2 -11989.508} C_VEL
LIN {X 0,Y 390.181,Z 671.834,A -85,B 0,C 180,E1 -11990.074,E2 -11990.074} C_VEL
LIN {X 0,Y 386.363,Z 639.716,A -85,B 0,C 180,E1 -11990.951,E2 -11990.951} C_VEL
LIN {X 0,Y 385.789,Z 635.091,A -85,B 0,C 180,E1 -11991.097,E2 -11991.097} C_VEL
LIN {X 0,Y 387.836,Z 609.108,A -85,B 0,C 180,E1 -11995.292,E2 -11995.292} C_VEL
LIN {X 0,Y 387.964,Z 604.486,A -85,B 0,C 180,E1 -11996.058,E2 -11996.058} C_VEL
LIN {X 0,Y 384.732,Z 589.802,A -85,B 0,C 180,E1 -11998.738,E2 -11998.738} C_VEL
LIN {X 0,Y 383.027,Z 582.773,A -85,B 0,C 180,E1 -12000.08,E2 -12000.08} C_VEL
LIN {X 0,Y 383.01,Z 582.776,A -85,B 0,C 180,E1 -12003.399,E2 -12003.399} C_VEL
LIN {X 0,Y 383.032,Z 582.775,A -85,B 0,C 180,E1 -12006.164,E2 -12006.164} C_VEL
LIN {X 0,Y 383.016,Z 582.776,A -85,B 0,C 180,E1 -12009.956,E2 -12009.956} C_VEL
LIN {X 0,Y 383.029,Z 582.771,A -85,B 0,C 180,E1 -12012.782,E2 -12012.782} C_VEL
LIN {X 0,Y 383.037,Z 582.766,A -85,B 0,C 180,E1 -12015.795,E2 -12015.795} C_VEL
LIN {X 0,Y 383.04,Z 582.768,A -85,B 0,C 180,E1 -12018.785,E2 -12018.785} C_VEL
LIN {X 0,Y 382.998,Z 582.776,A -85,B 0,C 180,E1 -12022.095,E2 -12022.095} C_VEL
LIN {X 0,Y 383.012,Z 582.761,A -85,B 0,C 180,E1 -12025.331,E2 -12025.331} C_VEL
LIN {X 0,Y 383.031,Z 582.771,A -85,B 0,C 180,E1 -12027.852,E2 -12027.852} C_VEL
LIN {X 0,Y 383.057,Z 582.756,A -85,B 0,C 180,E1 -12031.72,E2 -12031.72} C_VEL
LIN {X 0,Y 383.045,Z 582.767,A -85,B 0,C 180,E1 -12035.039,E2 -12035.039} C_VEL
LIN {X 0,Y 382.985,Z 582.769,A -85,B 0,C 180,E1 -12038.468,E2 -12038.468} C_VEL
LIN {X 0,Y 383.055,Z 582.767,A -85,B 0,C 180,E1 -12041.826,E2 -12041.826} C_VEL
LIN {X 0,Y 383.101,Z 582.756,A -85,B 0,C 180,E1 -12045.118,E2 -12045.118} C_VEL
LIN {X 0,Y 383.09,Z 582.767,A -85,B 0,C 180,E1 -12048.358,E2 -12048.358} C_VEL
LIN {X 0,Y 383.255,Z 582.729,A -85,B 0,C 180,E1 -12051.976,E2 -12051.976} C_VEL
LIN {X 0,Y 383.198,Z 582.754,A -85,B 0,C 180,E1 -12054.738,E2 -12054.738} C_VEL
LIN {X 0,Y 383.38,Z 582.715,A -85,B 0,C 180,E1 -12057.899,E2 -12057.899} C_VEL
LIN {X 0,Y 383.512,Z 582.703,A -85,B 0,C 180,E1 -12060,E2 -12060} C_VEL
LIN {X 0,Y 383.245,Z 582.742,A -85,B 0,C 180,E1 -12063.154,E2 -12063.154} C_VEL
LIN {X 0,Y 383.255,Z 582.73,A -85,B 0,C 180,E1 -12066.608,E2 -12066.608} C_VEL
LIN {X 0,Y 383.143,Z 582.756,A -85,B 0,C 180,E1 -12069.502,E2 -12069.502} C_VEL
LIN {X 0,Y 383.117,Z 582.755,A -85,B 0,C 180,E1 -12073.536,E2 -12073.536} C_VEL
LIN {X 0,Y 383.086,Z 582.758,A -85,B 0,C 180,E1 -12077.455,E2 -12077.455} C_VEL
LIN {X 0,Y 383.02,Z 582.769,A -85,B 0,C 180,E1 -12080.647,E2 -12080.647} C_VEL
LIN {X 0,Y 383.015,Z 582.765,A -85,B 0,C 180,E1 -12083.809,E2 -12083.809} C_VEL
LIN {X 0,Y 383.073,Z 582.762,A -85,B 0,C 180,E1 -12086.124,E2 -12086.124} C_VEL
LIN {X 0,Y 383.043,Z 582.77,A -85,B 0,C 180,E1 -12088.493,E2 -12088.493} C_VEL
LIN {X 0,Y 383.003,Z 582.775,A -85,B 0,C 180,E1 -12092.428,E2 -12092.428} C_VEL
LIN {X 0,Y 383.028,Z 582.771,A -85,B 0,C 180,E1 -12096.166,E2 -12096.166} C_VEL
LIN {X 0,Y 383.013,Z 582.769,A -85,B 0,C 180,E1 -12099.958,E2 -12099.958} C_VEL
LIN {X 0,Y 383.028,Z 582.75,A -85,B 0,C 180,E1 -12102.784,E2 -12102.784} C_VEL
LIN {X 0,Y 382.994,Z 582.775,A -85,B 0,C 180,E1 -12105.79,E2 -12105.79} C_VEL
LIN {X 0,Y 382.984,Z 582.77,A -85,B 0,C 180,E1 -12108.797,E2 -12108.797} C_VEL
LIN {X 0,Y 382.999,Z 582.766,A -85,B 0,C 180,E1 -12112.097,E2 -12112.097} C_VEL
LIN {X 0,Y 383.016,Z 582.777,A -85,B 0,C 180,E1 -12115.333,E2 -12115.333} C_VEL
LIN {X 0,Y 383.021,Z 582.774,A -85,B 0,C 180,E1 -12116.627,E2 -12116.627} C_VEL
LIN {X 0,Y 384.117,Z 585.783,A -85,B 0,C 180,E1 -12116.783,E2 -12116.783} C_VEL
LIN {X 0,Y 391.654,Z 602.615,A -85,B 0,C 180,E1 -12117.626,E2 -12117.626} C_VEL
LIN {X 0,Y 391.344,Z 628.449,A -85,B 0,C 180,E1 -12118.114,E2 -12118.114} C_VEL
LIN {X 0,Y 390.428,Z 682.369,A -85,B 0,C 180,E1 -12119.136,E2 -12119.136} C_VEL
LIN {X 0,Y 390.142,Z 695.086,A -85,B 0,C 180,E1 -12119.56,E2 -12119.56} C_VEL
LIN {X 0,Y 389.651,Z 707.139,A -85,B 0,C 180,E1 -12120.159,E2 -12120.159} C_VEL
LIN {X 0,Y 388.914,Z 718.79,A -85,B 0,C 180,E1 -12120.946,E2 -12120.946} C_VEL
LIN {X 0,Y 388.008,Z 729.849,A -85,B 0,C 180,E1 -12121.906,E2 -12121.906} C_VEL
LIN {X 0,Y 387.066,Z 739.959,A -85,B 0,C 180,E1 -12123.005,E2 -12123.005} C_VEL
LIN {X 0,Y 386.038,Z 750.06,A -85,B 0,C 180,E1 -12124.382,E2 -12124.382} C_VEL
LIN {X 0,Y 385.122,Z 758.684,A -85,B 0,C 180,E1 -12125.845,E2 -12125.845} C_VEL
LIN {X 0,Y 384.272,Z 766.162,A -85,B 0,C 180,E1 -12127.414,E2 -12127.414} C_VEL
LIN {X 0,Y 383.497,Z 772.731,A -85,B 0,C 180,E1 -12129.169,E2 -12129.169} C_VEL
LIN {X 0,Y 382.988,Z 777.26,A -85,B 0,C 180,E1 -12130.713,E2 -12130.713} C_VEL
LIN {X 0,Y 382.681,Z 779.852,A -85,B 0,C 180,E1 -12131.808,E2 -12131.808} C_VEL
LIN {X 0,Y 382.488,Z 781.926,A -85,B 0,C 180,E1 -12132.903,E2 -12132.903} C_VEL
LIN {X 0,Y 382.254,Z 783.541,A -85,B 0,C 180,E1 -12133.992,E2 -12133.992} C_VEL
LIN {X 0,Y 382.076,Z 784.744,A -85,B 0,C 180,E1 -12135.077,E2 -12135.077} C_VEL
LIN {X 0,Y 381.974,Z 785.499,A -85,B 0,C 180,E1 -12136.162,E2 -12136.162} C_VEL
LIN {X 0,Y 381.98,Z 785.828,A -85,B 0,C 180,E1 -12137.245,E2 -12137.245} C_VEL
LIN {X 0,Y 381.961,Z 785.774,A -85,B 0,C 180,E1 -12138.323,E2 -12138.323} C_VEL
LIN {X 0,Y 381.904,Z 785.326,A -85,B 0,C 180,E1 -12139.396,E2 -12139.396} C_VEL
LIN {X 0,Y 381.969,Z 784.43,A -85,B 0,C 180,E1 -12140.468,E2 -12140.468} C_VEL
LIN {X 0,Y 382.056,Z 783.146,A -85,B 0,C 180,E1 -12141.538,E2 -12141.538} C_VEL
LIN {X 0,Y 382.316,Z 780.573,A -85,B 0,C 180,E1 -12143.058,E2 -12143.058} C_VEL
LIN {X 0,Y 382.586,Z 776.684,A -85,B 0,C 180,E1 -12144.73,E2 -12144.73} C_VEL
LIN {X 0,Y 382.938,Z 771.847,A -85,B 0,C 180,E1 -12146.317,E2 -12146.317} C_VEL
LIN {X 0,Y 383.463,Z 765.752,A -85,B 0,C 180,E1 -12147.899,E2 -12147.899} C_VEL
LIN {X 0,Y 384.043,Z 758.128,A -85,B 0,C 180,E1 -12149.476,E2 -12149.476} C_VEL
LIN {X 0,Y 384.959,Z 748.608,A -85,B 0,C 180,E1 -12151.046,E2 -12151.046} C_VEL
LIN {X 0,Y 385.725,Z 738.729,A -85,B 0,C 180,E1 -12152.349,E2 -12152.349} C_VEL
LIN {X 0,Y 386.509,Z 727.665,A -85,B 0,C 180,E1 -12153.518,E2 -12153.518} C_VEL
LIN {X 0,Y 387.26,Z 716.809,A -85,B 0,C 180,E1 -12154.423,E2 -12154.423} C_VEL
LIN {X 0,Y 387.855,Z 704.687,A -85,B 0,C 180,E1 -12155.198,E2 -12155.198} C_VEL
LIN {X 0,Y 388.328,Z 691.371,A -85,B 0,C 180,E1 -12155.81,E2 -12155.81} C_VEL
LIN {X 0,Y 388.601,Z 679.275,A -85,B 0,C 180,E1 -12156.164,E2 -12156.164} C_VEL
LIN {X 0,Y 388.838,Z 659.957,A -85,B 0,C 180,E1 -12156.524,E2 -12156.524} C_VEL
LIN {X 0,Y 388.287,Z 654.144,A -85,B 0,C 180,E1 -12156.658,E2 -12156.658} C_VEL
LIN {X 0,Y 383.026,Z 635.426,A -85,B 0,C 180,E1 -12157.248,E2 -12157.248} C_VEL
LIN {X 0,Y 382.444,Z 629.614,A -85,B 0,C 180,E1 -12157.386,E2 -12157.386} C_VEL
LIN {X 0,Y 382.722,Z 601.725,A -85,B 0,C 180,E1 -12157.913,E2 -12157.913} C_VEL
LIN {X 0,Y 376.165,Z 583.629,A -85,B 0,C 180,E1 -12158.596,E2 -12158.596} C_VEL
LIN {X 0,Y 376.061,Z 583.643,A -85,B 0,C 180,E1 -12161.863,E2 -12161.863} C_VEL
LIN {X 0,Y 376.062,Z 583.639,A -85,B 0,C 180,E1 -12165.167,E2 -12165.167} C_VEL
LIN {X 0,Y 376.025,Z 583.645,A -85,B 0,C 180,E1 -12168.525,E2 -12168.525} C_VEL
LIN {X 0,Y 375.957,Z 583.656,A -85,B 0,C 180,E1 -12171.954,E2 -12171.954} C_VEL
LIN {X 0,Y 376.03,Z 583.643,A -85,B 0,C 180,E1 -12175.162,E2 -12175.162} C_VEL
LIN {X 0,Y 378.99,Z 591.62,A -85,B 0,C 180,E1 -12175.504,E2 -12175.504} C_VEL
LIN {X 0,Y 383.358,Z 603.233,A -85,B 0,C 180,E1 -12175.974,E2 -12175.974} C_VEL
LIN {X 0,Y 381.87,Z 684.028,A -85,B 0,C 180,E1 -12177.616,E2 -12177.616} C_VEL
LIN {X 0,Y 381.52,Z 697.536,A -85,B 0,C 180,E1 -12178.12,E2 -12178.12} C_VEL
LIN {X 0,Y 380.934,Z 710.239,A -85,B 0,C 180,E1 -12178.815,E2 -12178.815} C_VEL
LIN {X 0,Y 380.192,Z 723.049,A -85,B 0,C 180,E1 -12179.773,E2 -12179.773} C_VEL
LIN {X 0,Y 379.468,Z 733.506,A -85,B 0,C 180,E1 -12180.772,E2 -12180.772} C_VEL
LIN {X 0,Y 378.654,Z 743.633,A -85,B 0,C 180,E1 -12181.972,E2 -12181.972} C_VEL
LIN {X 0,Y 377.836,Z 752.761,A -85,B 0,C 180,E1 -12183.307,E2 -12183.307} C_VEL
LIN {X 0,Y 377.017,Z 761.569,A -85,B 0,C 180,E1 -12184.894,E2 -12184.894} C_VEL
LIN {X 0,Y 376.294,Z 768.991,A -85,B 0,C 180,E1 -12186.572,E2 -12186.572} C_VEL
LIN {X 0,Y 375.86,Z 774.823,A -85,B 0,C 180,E1 -12188.248,E2 -12188.248} C_VEL
LIN {X 0,Y 375.424,Z 779.244,A -85,B 0,C 180,E1 -12189.867,E2 -12189.867} C_VEL
LIN {X 0,Y 375.163,Z 782.538,A -85,B 0,C 180,E1 -12191.468,E2 -12191.468} C_VEL
LIN {X 0,Y 374.926,Z 784.823,A -85,B 0,C 180,E1 -12193.025,E2 -12193.025} C_VEL
LIN {X 0,Y 374.819,Z 786.231,A -85,B 0,C 180,E1 -12194.56,E2 -12194.56} C_VEL
LIN {X 0,Y 374.811,Z 786.786,A -85,B 0,C 180,E1 -12196.07,E2 -12196.07} C_VEL
LIN {X 0,Y 374.879,Z 786.562,A -85,B 0,C 180,E1 -12197.553,E2 -12197.553} C_VEL
LIN {X 0,Y 374.983,Z 785.628,A -85,B 0,C 180,E1 -12199.006,E2 -12199.006} C_VEL
LIN {X 0,Y 375.21,Z 783.973,A -85,B 0,C 180,E1 -12200.443,E2 -12200.443} C_VEL
LIN {X 0,Y 375.707,Z 780.082,A -85,B 0,C 180,E1 -12202.559,E2 -12202.559} C_VEL
LIN {X 0,Y 376.088,Z 776.256,A -85,B 0,C 180,E1 -12204.059,E2 -12204.059} C_VEL
LIN {X 0,Y 376.764,Z 769.904,A -85,B 0,C 180,E1 -12205.971,E2 -12205.971} C_VEL
LIN {X 0,Y 377.607,Z 762.65,A -85,B 0,C 180,E1 -12207.65,E2 -12207.65} C_VEL
LIN {X 0,Y 378.618,Z 753.614,A -85,B 0,C 180,E1 -12209.305,E2 -12209.305} C_VEL
LIN {X 0,Y 379.434,Z 745.448,A -85,B 0,C 180,E1 -12210.52,E2 -12210.52} C_VEL
LIN {X 0,Y 380.363,Z 735.721,A -85,B 0,C 180,E1 -12211.71,E2 -12211.71} C_VEL
LIN {X 0,Y 381.202,Z 725.657,A -85,B 0,C 180,E1 -12212.703,E2 -12212.703} C_VEL
LIN {X 0,Y 381.998,Z 713.472,A -85,B 0,C 180,E1 -12213.65,E2 -12213.65} C_VEL
LIN {X 0,Y 382.64,Z 701.266,A -85,B 0,C 180,E1 -12214.364,E2 -12214.364} C_VEL
LIN {X 0,Y 382.961,Z 688.455,A -85,B 0,C 180,E1 -12214.889,E2 -12214.889} C_VEL
LIN {X 0,Y 383.342,Z 669.564,A -85,B 0,C 180,E1 -12215.332,E2 -12215.332} C_VEL
LIN {X 0,Y 384.717,Z 603.91,A -85,B 0,C 180,E1 -12216.679,E2 -12216.679} C_VEL
LIN {X 0,Y 376.974,Z 586.504,A -85,B 0,C 180,E1 -12217.603,E2 -12217.603} C_VEL
LIN {X 0,Y 375.946,Z 583.656,A -85,B 0,C 180,E1 -12217.756,E2 -12217.756} C_VEL
LIN {X 0,Y 375.99,Z 583.653,A -85,B 0,C 180,E1 -12220.339,E2 -12220.339} C_VEL
LIN {X 0,Y 376.021,Z 583.646,A -85,B 0,C 180,E1 -12223.718,E2 -12223.718} C_VEL
LIN {X 0,Y 376.099,Z 583.638,A -85,B 0,C 180,E1 -12227.042,E2 -12227.042} C_VEL
LIN {X 0,Y 376.116,Z 583.634,A -85,B 0,C 180,E1 -12230.318,E2 -12230.318} C_VEL
LIN {X 0,Y 376.222,Z 583.621,A -85,B 0,C 180,E1 -12232.486,E2 -12232.486} C_VEL
LIN {X 0,Y 376.17,Z 583.627,A -85,B 0,C 180,E1 -12234.64,E2 -12234.64} C_VEL
LIN {X 0,Y 376.346,Z 583.601,A -85,B 0,C 180,E1 -12237.86,E2 -12237.86} C_VEL
LIN {X 0,Y 376.482,Z 583.589,A -85,B 0,C 180,E1 -12240,E2 -12240} C_VEL
LIN {X 0,Y 376.183,Z 583.62,A -85,B 0,C 180,E1 -12243.213,E2 -12243.213} C_VEL
LIN {X 0,Y 376.241,Z 583.615,A -85,B 0,C 180,E1 -12246.435,E2 -12246.435} C_VEL
LIN {X 0,Y 376.115,Z 583.628,A -85,B 0,C 180,E1 -12249.682,E2 -12249.682} C_VEL
LIN {X 0,Y 376.082,Z 583.626,A -85,B 0,C 180,E1 -12253.658,E2 -12253.658} C_VEL
LIN {X 0,Y 376.036,Z 583.635,A -85,B 0,C 180,E1 -12257.608,E2 -12257.608} C_VEL
LIN {X 0,Y 375.971,Z 583.647,A -85,B 0,C 180,E1 -12260.833,E2 -12260.833} C_VEL
LIN {X 0,Y 375.987,Z 583.645,A -85,B 0,C 180,E1 -12264.282,E2 -12264.282} C_VEL
LIN {X 0,Y 376.013,Z 583.644,A -85,B 0,C 180,E1 -12266.653,E2 -12266.653} C_VEL
LIN {X 0,Y 375.97,Z 583.652,A -85,B 0,C 180,E1 -12269.079,E2 -12269.079} C_VEL
LIN {X 0,Y 375.949,Z 583.653,A -85,B 0,C 180,E1 -12272.829,E2 -12272.829} C_VEL
LIN {X 0,Y 375.953,Z 583.653,A -85,B 0,C 180,E1 -12275.416,E2 -12275.416} C_VEL
LIN {X 0,Y 375.973,Z 583.655,A -85,B 0,C 180,E1 -12278.272,E2 -12278.272} C_VEL
LIN {X 0,Y 375.985,Z 583.647,A -85,B 0,C 180,E1 -12281.611,E2 -12281.611} C_VEL
LIN {X 0,Y 375.965,Z 583.653,A -85,B 0,C 180,E1 -12285.263,E2 -12285.263} C_VEL
LIN {X 0,Y 375.978,Z 583.651,A -85,B 0,C 180,E1 -12289.139,E2 -12289.139} C_VEL
LIN {X 0,Y 375.965,Z 583.654,A -85,B 0,C 180,E1 -12291.913,E2 -12291.913} C_VEL
LIN {X 0,Y 375.978,Z 583.65,A -85,B 0,C 180,E1 -12295.333,E2 -12295.333} C_VEL
LIN {X 0,Y 375.969,Z 583.836,A -85,B 0,C 180,E1 -12297.532,E2 -12297.532} C_VEL
LIN {X 0,Y 378.859,Z 595.884,A -85,B 0,C 180,E1 -12300.372,E2 -12300.372} C_VEL
LIN {X 0,Y 380.82,Z 605.577,A -85,B 0,C 180,E1 -12302.525,E2 -12302.525} C_VEL
LIN {X 0,Y 380.551,Z 611.408,A -85,B 0,C 180,E1 -12303.691,E2 -12303.691} C_VEL
LIN {X 0,Y 378.502,Z 633.281,A -85,B 0,C 180,E1 -12307.914,E2 -12307.914} C_VEL
LIN {X 0,Y 378.349,Z 635.568,A -85,B 0,C 180,E1 -12308.346,E2 -12308.346} C_VEL
LIN {X 0,Y 382.106,Z 661.289,A -85,B 0,C 180,E1 -12309.159,E2 -12309.159} C_VEL
LIN {X 0,Y 383.71,Z 677.061,A -85,B 0,C 180,E1 -12309.601,E2 -12309.601} C_VEL
LIN {X 0,Y 382.396,Z 746.082,A -85,B 0,C 180,E1 -12311.03,E2 -12311.03} C_VEL
LIN {X 0,Y 381.628,Z 759.744,A -85,B 0,C 180,E1 -12311.513,E2 -12311.513} C_VEL
LIN {X 0,Y 380.668,Z 772.767,A -85,B 0,C 180,E1 -12312.195,E2 -12312.195} C_VEL
LIN {X 0,Y 379.692,Z 784.678,A -85,B 0,C 180,E1 -12313.051,E2 -12313.051} C_VEL
LIN {X 0,Y 378.549,Z 796.199,A -85,B 0,C 180,E1 -12314.107,E2 -12314.107} C_VEL
LIN {X 0,Y 377.574,Z 806.955,A -85,B 0,C 180,E1 -12315.35,E2 -12315.35} C_VEL
LIN {X 0,Y 376.824,Z 815.235,A -85,B 0,C 180,E1 -12316.519,E2 -12316.519} C_VEL
LIN {X 0,Y 375.898,Z 824.576,A -85,B 0,C 180,E1 -12318.132,E2 -12318.132} C_VEL
LIN {X 0,Y 375.28,Z 832.148,A -85,B 0,C 180,E1 -12319.752,E2 -12319.752} C_VEL
LIN {X 0,Y 374.968,Z 838.254,A -85,B 0,C 180,E1 -12321.377,E2 -12321.377} C_VEL
LIN {X 0,Y 374.816,Z 843.091,A -85,B 0,C 180,E1 -12323,E2 -12323} C_VEL
LIN {X 0,Y 374.759,Z 846.802,A -85,B 0,C 180,E1 -12324.62,E2 -12324.62} C_VEL
LIN {X 0,Y 374.702,Z 848.681,A -85,B 0,C 180,E1 -12325.697,E2 -12325.697} C_VEL
LIN {X 0,Y 374.827,Z 850.134,A -85,B 0,C 180,E1 -12326.775,E2 -12326.775} C_VEL
LIN {X 0,Y 374.875,Z 851.171,A -85,B 0,C 180,E1 -12327.851,E2 -12327.851} C_VEL
LIN {X 0,Y 374.903,Z 851.795,A -85,B 0,C 180,E1 -12328.926,E2 -12328.926} C_VEL
LIN {X 0,Y 374.867,Z 851.959,A -85,B 0,C 180,E1 -12330,E2 -12330} C_VEL
LIN {X 0,Y 374.905,Z 851.721,A -85,B 0,C 180,E1 -12331.074,E2 -12331.074} C_VEL
LIN {X 0,Y 374.897,Z 851.074,A -85,B 0,C 180,E1 -12332.149,E2 -12332.149} C_VEL
LIN {X 0,Y 374.848,Z 850.007,A -85,B 0,C 180,E1 -12333.224,E2 -12333.224} C_VEL
LIN {X 0,Y 374.714,Z 848.456,A -85,B 0,C 180,E1 -12334.302,E2 -12334.302} C_VEL
LIN {X 0,Y 374.744,Z 845.255,A -85,B 0,C 180,E1 -12335.953,E2 -12335.953} C_VEL
LIN {X 0,Y 374.811,Z 841.101,A -85,B 0,C 180,E1 -12337.542,E2 -12337.542} C_VEL
LIN {X 0,Y 375.157,Z 833.721,A -85,B 0,C 180,E1 -12339.706,E2 -12339.706} C_VEL
LIN {X 0,Y 375.67,Z 826.947,A -85,B 0,C 180,E1 -12341.328,E2 -12341.328} C_VEL
LIN {X 0,Y 376.418,Z 818.567,A -85,B 0,C 180,E1 -12342.947,E2 -12342.947} C_VEL
LIN {X 0,Y 377.365,Z 808.916,A -85,B 0,C 180,E1 -12344.432,E2 -12344.432} C_VEL
LIN {X 0,Y 378.352,Z 799.351,A -85,B 0,C 180,E1 -12345.625,E2 -12345.625} C_VEL
LIN {X 0,Y 379.436,Z 788.847,A -85,B 0,C 180,E1 -12346.684,E2 -12346.684} C_VEL
LIN {X 0,Y 380.504,Z 777.18,A -85,B 0,C 180,E1 -12347.604,E2 -12347.604} C_VEL
LIN {X 0,Y 381.436,Z 765.073,A -85,B 0,C 180,E1 -12348.323,E2 -12348.323} C_VEL
LIN {X 0,Y 382.288,Z 751.835,A -85,B 0,C 180,E1 -12348.871,E2 -12348.871} C_VEL
LIN {X 0,Y 382.706,Z 736.93,A -85,B 0,C 180,E1 -12349.232,E2 -12349.232} C_VEL
LIN {X 0,Y 383.65,Z 672.705,A -85,B 0,C 180,E1 -12350.462,E2 -12350.462} C_VEL
LIN {X 0,Y 380.005,Z 641.541,A -85,B 0,C 180,E1 -12351.332,E2 -12351.332} C_VEL
LIN {X 0,Y 378.964,Z 633.837,A -85,B 0,C 180,E1 -12351.575,E2 -12351.575} C_VEL
LIN {X 0,Y 381.022,Z 608.861,A -85,B 0,C 180,E1 -12355.686,E2 -12355.686} C_VEL
LIN {X 0,Y 380.947,Z 605.397,A -85,B 0,C 180,E1 -12356.28,E2 -12356.28} C_VEL
LIN {X 0,Y 377.79,Z 591.182,A -85,B 0,C 180,E1 -12358.925,E2 -12358.925} C_VEL
LIN {X 0,Y 375.969,Z 583.654,A -85,B 0,C 180,E1 -12360.381,E2 -12360.381} C_VEL
LIN {X 0,Y 375.961,Z 583.656,A -85,B 0,C 180,E1 -12364.11,E2 -12364.11} C_VEL
LIN {X 0,Y 375.953,Z 583.654,A -85,B 0,C 180,E1 -12366.74,E2 -12366.74} C_VEL
LIN {X 0,Y 375.995,Z 583.651,A -85,B 0,C 180,E1 -12369.972,E2 -12369.972} C_VEL
LIN {X 0,Y 375.942,Z 583.656,A -85,B 0,C 180,E1 -12373.763,E2 -12373.763} C_VEL
LIN {X 0,Y 375.986,Z 583.648,A -85,B 0,C 180,E1 -12376.801,E2 -12376.801} C_VEL
LIN {X 0,Y 375.995,Z 583.642,A -85,B 0,C 180,E1 -12380.027,E2 -12380.027} C_VEL
LIN {X 0,Y 375.96,Z 583.651,A -85,B 0,C 180,E1 -12383.494,E2 -12383.494} C_VEL
LIN {X 0,Y 375.955,Z 583.642,A -85,B 0,C 180,E1 -12385.888,E2 -12385.888} C_VEL
LIN {X 0,Y 375.963,Z 583.649,A -85,B 0,C 180,E1 -12389.687,E2 -12389.687} C_VEL
LIN {X 0,Y 375.995,Z 583.639,A -85,B 0,C 180,E1 -12392.141,E2 -12392.141} C_VEL
LIN {X 0,Y 375.999,Z 583.649,A -85,B 0,C 180,E1 -12394.538,E2 -12394.538} C_VEL
LIN {X 0,Y 375.955,Z 583.639,A -85,B 0,C 180,E1 -12398.045,E2 -12398.045} C_VEL
LIN {X 0,Y 376.001,Z 583.645,A -85,B 0,C 180,E1 -12401.473,E2 -12401.473} C_VEL
LIN {X 0,Y 376.05,Z 583.631,A -85,B 0,C 180,E1 -12404.832,E2 -12404.832} C_VEL
LIN {X 0,Y 376.042,Z 583.643,A -85,B 0,C 180,E1 -12408.136,E2 -12408.136} C_VEL
LIN {X 0,Y 376.21,Z 583.606,A -85,B 0,C 180,E1 -12411.919,E2 -12411.919} C_VEL
LIN {X 0,Y 376.169,Z 583.63,A -85,B 0,C 180,E1 -12414.64,E2 -12414.64} C_VEL
LIN {X 0,Y 376.346,Z 583.591,A -85,B 0,C 180,E1 -12417.86,E2 -12417.86} C_VEL
LIN {X 0,Y 376.482,Z 583.579,A -85,B 0,C 180,E1 -12420,E2 -12420} C_VEL
LIN {X 0,Y 376.183,Z 583.621,A -85,B 0,C 180,E1 -12423.213,E2 -12423.213} C_VEL
LIN {X 0,Y 376.22,Z 583.605,A -85,B 0,C 180,E1 -12426.596,E2 -12426.596} C_VEL
LIN {X 0,Y 376.111,Z 583.632,A -85,B 0,C 180,E1 -12429.682,E2 -12429.682} C_VEL
LIN {X 0,Y 376.081,Z 583.631,A -85,B 0,C 180,E1 -12433.658,E2 -12433.658} C_VEL
LIN {X 0,Y 376.036,Z 583.635,A -85,B 0,C 180,E1 -12437.608,E2 -12437.608} C_VEL
LIN {X 0,Y 375.971,Z 583.649,A -85,B 0,C 180,E1 -12440.833,E2 -12440.833} C_VEL
LIN {X 0,Y 375.981,Z 583.642,A -85,B 0,C 180,E1 -12444.282,E2 -12444.282} C_VEL
LIN {X 0,Y 376.013,Z 583.644,A -85,B 0,C 180,E1 -12446.653,E2 -12446.653} C_VEL
LIN {X 0,Y 375.97,Z 583.646,A -85,B 0,C 180,E1 -12449.079,E2 -12449.079} C_VEL
LIN {X 0,Y 375.95,Z 583.656,A -85,B 0,C 180,E1 -12452.829,E2 -12452.829} C_VEL
LIN {X 0,Y 375.952,Z 583.653,A -85,B 0,C 180,E1 -12455.416,E2 -12455.416} C_VEL
LIN {X 0,Y 375.972,Z 583.65,A -85,B 0,C 180,E1 -12458.272,E2 -12458.272} C_VEL
LIN {X 0,Y 375.955,Z 583.63,A -85,B 0,C 180,E1 -12461.606,E2 -12461.606} C_VEL
LIN {X 0,Y 375.95,Z 583.658,A -85,B 0,C 180,E1 -12465.265,E2 -12465.265} C_VEL
LIN {X 0,Y 375.937,Z 583.651,A -85,B 0,C 180,E1 -12469.134,E2 -12469.134} C_VEL
LIN {X 0,Y 375.963,Z 583.642,A -85,B 0,C 180,E1 -12471.913,E2 -12471.913} C_VEL
LIN {X 0,Y 375.978,Z 583.654,A -85,B 0,C 180,E1 -12475.333,E2 -12475.333} C_VEL
LIN {X 0,Y 375.963,Z 583.668,A -85,B 0,C 180,E1 -12476.159,E2 -12476.159} C_VEL
LIN {X 0,Y 376.978,Z 586.488,A -85,B 0,C 180,E1 -12476.292,E2 -12476.292} C_VEL
LIN {X 0,Y 384.703,Z 603.333,A -85,B 0,C 180,E1 -12477.178,E2 -12477.178} C_VEL
LIN {X 0,Y 385.307,Z 604.86,A -85,B 0,C 180,E1 -12477.25,E2 -12477.25} C_VEL
LIN {X 0,Y 383.889,Z 682.937,A -85,B 0,C 180,E1 -12478.742,E2 -12478.742} C_VEL
LIN {X 0,Y 383.535,Z 696.571,A -85,B 0,C 180,E1 -12479.21,E2 -12479.21} C_VEL
LIN {X 0,Y 383.024,Z 708.263,A -85,B 0,C 180,E1 -12479.815,E2 -12479.815} C_VEL
LIN {X 0,Y 382.316,Z 718.936,A -85,B 0,C 180,E1 -12480.546,E2 -12480.546} C_VEL
LIN {X 0,Y 381.363,Z 730.077,A -85,B 0,C 180,E1 -12481.522,E2 -12481.522} C_VEL
LIN {X 0,Y 380.408,Z 739.908,A -85,B 0,C 180,E1 -12482.599,E2 -12482.599} C_VEL
LIN {X 0,Y 379.402,Z 749.527,A -85,B 0,C 180,E1 -12483.901,E2 -12483.901} C_VEL
LIN {X 0,Y 378.505,Z 757.509,A -85,B 0,C 180,E1 -12485.232,E2 -12485.232} C_VEL
LIN {X 0,Y 377.466,Z 765.994,A -85,B 0,C 180,E1 -12486.984,E2 -12486.984} C_VEL
LIN {X 0,Y 376.72,Z 772.213,A -85,B 0,C 180,E1 -12488.604,E2 -12488.604} C_VEL
LIN {X 0,Y 376.054,Z 777.416,A -85,B 0,C 180,E1 -12490.343,E2 -12490.343} C_VEL
LIN {X 0,Y 375.591,Z 781.208,A -85,B 0,C 180,E1 -12492.017,E2 -12492.017} C_VEL
LIN {X 0,Y 375.248,Z 783.921,A -85,B 0,C 180,E1 -12493.684,E2 -12493.684} C_VEL
LIN {X 0,Y 375.06,Z 785.175,A -85,B 0,C 180,E1 -12494.792,E2 -12494.792} C_VEL
LIN {X 0,Y 374.942,Z 786.023,A -85,B 0,C 180,E1 -12495.897,E2 -12495.897} C_VEL
LIN {X 0,Y 374.902,Z 786.427,A -85,B 0,C 180,E1 -12497.112,E2 -12497.112} C_VEL
LIN {X 0,Y 374.832,Z 786.023,A -85,B 0,C 180,E1 -12499.193,E2 -12499.193} C_VEL
LIN {X 0,Y 374.881,Z 785.213,A -85,B 0,C 180,E1 -12500.287,E2 -12500.287} C_VEL
LIN {X 0,Y 374.982,Z 783.976,A -85,B 0,C 180,E1 -12501.377,E2 -12501.377} C_VEL
LIN {X 0,Y 375.239,Z 781.26,A -85,B 0,C 180,E1 -12503.054,E2 -12503.054} C_VEL
LIN {X 0,Y 375.481,Z 777.729,A -85,B 0,C 180,E1 -12504.63,E2 -12504.63} C_VEL
LIN {X 0,Y 375.848,Z 773.006,A -85,B 0,C 180,E1 -12506.248,E2 -12506.248} C_VEL
LIN {X 0,Y 376.364,Z 767.045,A -85,B 0,C 180,E1 -12507.86,E2 -12507.86} C_VEL
LIN {X 0,Y 376.986,Z 759.632,A -85,B 0,C 180,E1 -12509.466,E2 -12509.466} C_VEL
LIN {X 0,Y 377.914,Z 750.289,A -85,B 0,C 180,E1 -12511.066,E2 -12511.066} C_VEL
LIN {X 0,Y 378.712,Z 740.713,A -85,B 0,C 180,E1 -12512.393,E2 -12512.393} C_VEL
LIN {X 0,Y 379.494,Z 729.969,A -85,B 0,C 180,E1 -12513.583,E2 -12513.583} C_VEL
LIN {X 0,Y 380.368,Z 717.842,A -85,B 0,C 180,E1 -12514.637,E2 -12514.637} C_VEL
LIN {X 0,Y 381.001,Z 705.892,A -85,B 0,C 180,E1 -12515.424,E2 -12515.424} C_VEL
LIN {X 0,Y 381.479,Z 692.804,A -85,B 0,C 180,E1 -12516.048,E2 -12516.048} C_VEL
LIN {X 0,Y 381.783,Z 679.917,A -85,B 0,C 180,E1 -12516.441,E2 -12516.441} C_VEL
LIN {X 0,Y 382.444,Z 629.614,A -85,B 0,C 180,E1 -12517.386,E2 -12517.386} C_VEL
LIN {X 0,Y 381.759,Z 621.842,A -85,B 0,C 180,E1 -12517.568,E2 -12517.568} C_VEL
LIN {X 0,Y 379.925,Z 614.291,A -85,B 0,C 180,E1 -12517.8,E2 -12517.8} C_VEL
LIN {X 0,Y 374.627,Z 599.609,A -85,B 0,C 180,E1 -12518.341,E2 -12518.341} C_VEL
LIN {X 0,Y 369.105,Z 584.507,A -85,B 0,C 180,E1 -12518.933,E2 -12518.933} C_VEL
LIN {X 0,Y 369.015,Z 584.522,A -85,B 0,C 180,E1 -12522.093,E2 -12522.093} C_VEL
LIN {X 0,Y 369.001,Z 584.519,A -85,B 0,C 180,E1 -12525.464,E2 -12525.464} C_VEL
LIN {X 0,Y 368.984,Z 584.521,A -85,B 0,C 180,E1 -12528.892,E2 -12528.892} C_VEL
LIN {X 0,Y 368.923,Z 584.53,A -85,B 0,C 180,E1 -12532.395,E2 -12532.395} C_VEL
LIN {X 0,Y 368.973,Z 584.526,A -85,B 0,C 180,E1 -12534.811,E2 -12534.811} C_VEL
LIN {X 0,Y 372.505,Z 593.902,A -85,B 0,C 180,E1 -12535.21,E2 -12535.21} C_VEL
LIN {X 0,Y 376.627,Z 604.574,A -85,B 0,C 180,E1 -12535.66,E2 -12535.66} C_VEL
LIN {X 0,Y 375.082,Z 684.262,A -85,B 0,C 180,E1 -12537.307,E2 -12537.307} C_VEL
LIN {X 0,Y 374.721,Z 697.629,A -85,B 0,C 180,E1 -12537.809,E2 -12537.809} C_VEL
LIN {X 0,Y 374.185,Z 709.914,A -85,B 0,C 180,E1 -12538.48,E2 -12538.48} C_VEL
LIN {X 0,Y 373.399,Z 722.429,A -85,B 0,C 180,E1 -12539.41,E2 -12539.41} C_VEL
LIN {X 0,Y 372.67,Z 733.046,A -85,B 0,C 180,E1 -12540.422,E2 -12540.422} C_VEL
LIN {X 0,Y 371.754,Z 743.913,A -85,B 0,C 180,E1 -12541.709,E2 -12541.709} C_VEL
LIN {X 0,Y 370.865,Z 753.725,A -85,B 0,C 180,E1 -12543.173,E2 -12543.173} C_VEL
LIN {X 0,Y 370.023,Z 762.212,A -85,B 0,C 180,E1 -12544.735,E2 -12544.735} C_VEL
LIN {X 0,Y 369.407,Z 768.423,A -85,B 0,C 180,E1 -12546.14,E2 -12546.14} C_VEL
LIN {X 0,Y 369.02,Z 773.541,A -85,B 0,C 180,E1 -12547.548,E2 -12547.548} C_VEL
LIN {X 0,Y 368.596,Z 777.844,A -85,B 0,C 180,E1 -12548.991,E2 -12548.991} C_VEL
LIN {X 0,Y 368.258,Z 781.327,A -85,B 0,C 180,E1 -12550.455,E2 -12550.455} C_VEL
LIN {X 0,Y 368.01,Z 784.026,A -85,B 0,C 180,E1 -12551.943,E2 -12551.943} C_VEL
LIN {X 0,Y 367.832,Z 785.927,A -85,B 0,C 180,E1 -12553.458,E2 -12553.458} C_VEL
LIN {X 0,Y 367.742,Z 787.064,A -85,B 0,C 180,E1 -12554.999,E2 -12554.999} C_VEL
LIN {X 0,Y 367.759,Z 787.418,A -85,B 0,C 180,E1 -12556.567,E2 -12556.567} C_VEL
LIN {X 0,Y 367.841,Z 786.942,A -85,B 0,C 180,E1 -12558.169,E2 -12558.169} C_VEL
LIN {X 0,Y 368.033,Z 785.566,A -85,B 0,C 180,E1 -12559.803,E2 -12559.803} C_VEL
LIN {X 0,Y 368.397,Z 783.211,A -85,B 0,C 180,E1 -12561.458,E2 -12561.458} C_VEL
LIN {X 0,Y 368.818,Z 779.735,A -85,B 0,C 180,E1 -12563.16,E2 -12563.16} C_VEL
LIN {X 0,Y 369.434,Z 773.994,A -85,B 0,C 180,E1 -12565.2,E2 -12565.2} C_VEL
LIN {X 0,Y 370.266,Z 767.371,A -85,B 0,C 180,E1 -12566.993,E2 -12566.993} C_VEL
LIN {X 0,Y 371.121,Z 759.955,A -85,B 0,C 180,E1 -12568.576,E2 -12568.576} C_VEL
LIN {X 0,Y 372.152,Z 750.958,A -85,B 0,C 180,E1 -12570.119,E2 -12570.119} C_VEL
LIN {X 0,Y 373.17,Z 741.343,A -85,B 0,C 180,E1 -12571.452,E2 -12571.452} C_VEL
LIN {X 0,Y 374.075,Z 731.125,A -85,B 0,C 180,E1 -12572.594,E2 -12572.594} C_VEL
LIN {X 0,Y 374.974,Z 719.646,A -85,B 0,C 180,E1 -12573.608,E2 -12573.608} C_VEL
LIN {X 0,Y 375.803,Z 707.33,A -85,B 0,C 180,E1 -12574.442,E2 -12574.442} C_VEL
LIN {X 0,Y 376.255,Z 694.439,A -85,B 0,C 180,E1 -12575.074,E2 -12575.074} C_VEL
LIN {X 0,Y 376.578,Z 681.447,A -85,B 0,C 180,E1 -12575.483,E2 -12575.483} C_VEL
LIN {X 0,Y 378.234,Z 605.831,A -85,B 0,C 180,E1 -12577.069,E2 -12577.069} C_VEL
LIN {X 0,Y 371.261,Z 590.194,A -85,B 0,C 180,E1 -12577.934,E2 -12577.934} C_VEL
LIN {X 0,Y 369.114,Z 585.479,A -85,B 0,C 180,E1 -12578.206,E2 -12578.206} C_VEL
LIN {X 0,Y 368.907,Z 584.531,A -85,B 0,C 180,E1 -12578.266,E2 -12578.266} C_VEL
LIN {X 0,Y 368.95,Z 584.529,A -85,B 0,C 180,E1 -12581.105,E2 -12581.105} C_VEL
LIN {X 0,Y 368.99,Z 584.524,A -85,B 0,C 180,E1 -12584.535,E2 -12584.535} C_VEL
LIN {X 0,Y 369.006,Z 584.521,A -85,B 0,C 180,E1 -12587.907,E2 -12587.907} C_VEL
LIN {X 0,Y 369.221,Z 584.493,A -85,B 0,C 180,E1 -12591.801,E2 -12591.801} C_VEL
LIN {X 0,Y 369.142,Z 584.503,A -85,B 0,C 180,E1 -12594.538,E2 -12594.538} C_VEL
LIN {X 0,Y 369.311,Z 584.477,A -85,B 0,C 180,E1 -12597.819,E2 -12597.819} C_VEL
LIN {X 0,Y 369.451,Z 584.464,A -85,B 0,C 180,E1 -12600,E2 -12600} C_VEL
LIN {X 0,Y 369.31,Z 584.483,A -85,B 0,C 180,E1 -12602.181,E2 -12602.181} C_VEL
LIN {X 0,Y 369.2,Z 584.491,A -85,B 0,C 180,E1 -12606.558,E2 -12606.558} C_VEL
LIN {X 0,Y 369.114,Z 584.504,A -85,B 0,C 180,E1 -12608.762,E2 -12608.762} C_VEL
LIN {X 0,Y 369.005,Z 584.516,A -85,B 0,C 180,E1 -12612.093,E2 -12612.093} C_VEL
LIN {X 0,Y 368.99,Z 584.515,A -85,B 0,C 180,E1 -12615.465,E2 -12615.465} C_VEL
LIN {X 0,Y 368.975,Z 584.52,A -85,B 0,C 180,E1 -12618.893,E2 -12618.893} C_VEL
LIN {X 0,Y 368.925,Z 584.53,A -85,B 0,C 180,E1 -12622.396,E2 -12622.396} C_VEL
LIN {X 0,Y 368.993,Z 584.521,A -85,B 0,C 180,E1 -12625.981,E2 -12625.981} C_VEL
LIN {X 0,Y 368.961,Z 584.527,A -85,B 0,C 180,E1 -12628.814,E2 -12628.814} C_VEL
LIN {X 0,Y 368.897,Z 584.535,A -85,B 0,C 180,E1 -12632.238,E2 -12632.238} C_VEL
LIN {X 0,Y 368.924,Z 584.531,A -85,B 0,C 180,E1 -12635.002,E2 -12635.002} C_VEL
LIN {X 0,Y 368.908,Z 584.531,A -85,B 0,C 180,E1 -12638.642,E2 -12638.642} C_VEL
LIN {X 0,Y 368.938,Z 584.526,A -85,B 0,C 180,E1 -12642.021,E2 -12642.021} C_VEL
LIN {X 0,Y 368.919,Z 584.531,A -85,B 0,C 180,E1 -12645.183,E2 -12645.183} C_VEL
LIN {X 0,Y 368.907,Z 584.534,A -85,B 0,C 180,E1 -12648.182,E2 -12648.182} C_VEL
LIN {X 0,Y 368.91,Z 584.532,A -85,B 0,C 180,E1 -12651.36,E2 -12651.36} C_VEL
LIN {X 0,Y 368.935,Z 584.527,A -85,B 0,C 180,E1 -12655.147,E2 -12655.147} C_VEL
LIN {X 0,Y 368.936,Z 584.644,A -85,B 0,C 180,E1 -12657.057,E2 -12657.057} C_VEL
LIN {X 0,Y 371.777,Z 596.339,A -85,B 0,C 180,E1 -12659.903,E2 -12659.903} C_VEL
LIN {X 0,Y 373.916,Z 606.931,A -85,B 0,C 180,E1 -12662.325,E2 -12662.325} C_VEL
LIN {X 0,Y 373.809,Z 611.06,A -85,B 0,C 180,E1 -12663.178,E2 -12663.178} C_VEL
LIN {X 0,Y 371.962,Z 629.966,A -85,B 0,C 180,E1 -12666.918,E2 -12666.918} C_VEL
LIN {X 0,Y 371.51,Z 634.768,A -85,B 0,C 180,E1 -12667.856,E2 -12667.856} C_VEL
LIN {X 0,Y 374.867,Z 656.585,A -85,B 0,C 180,E1 -12668.592,E2 -12668.592} C_VEL
LIN {X 0,Y 377.132,Z 676.208,A -85,B 0,C 180,E1 -12669.175,E2 -12669.175} C_VEL
LIN {X 0,Y 375.768,Z 745.646,A -85,B 0,C 180,E1 -12670.647,E2 -12670.647} C_VEL
LIN {X 0,Y 374.976,Z 759.203,A -85,B 0,C 180,E1 -12671.137,E2 -12671.137} C_VEL
LIN {X 0,Y 374.013,Z 771.62,A -85,B 0,C 180,E1 -12671.797,E2 -12671.797} C_VEL
LIN {X 0,Y 373.025,Z 782.824,A -85,B 0,C 180,E1 -12672.597,E2 -12672.597} C_VEL
LIN {X 0,Y 371.849,Z 794.534,A -85,B 0,C 180,E1 -12673.672,E2 -12673.672} C_VEL
LIN {X 0,Y 370.812,Z 805.022,A -85,B 0,C 180,E1 -12674.879,E2 -12674.879} C_VEL
LIN {X 0,Y 369.902,Z 814.764,A -85,B 0,C 180,E1 -12676.262,E2 -12676.262} C_VEL
LIN {X 0,Y 369.064,Z 822.68,A -85,B 0,C 180,E1 -12677.63,E2 -12677.63} C_VEL
LIN {X 0,Y 368.313,Z 830.466,A -85,B 0,C 180,E1 -12679.278,E2 -12679.278} C_VEL
LIN {X 0,Y 367.979,Z 835.818,A -85,B 0,C 180,E1 -12680.657,E2 -12680.657} C_VEL
LIN {X 0,Y 367.765,Z 841.034,A -85,B 0,C 180,E1 -12682.313,E2 -12682.313} C_VEL
LIN {X 0,Y 367.679,Z 844.535,A -85,B 0,C 180,E1 -12683.698,E2 -12683.698} C_VEL
LIN {X 0,Y 367.627,Z 848.094,A -85,B 0,C 180,E1 -12685.614,E2 -12685.614} C_VEL
LIN {X 0,Y 367.73,Z 849.537,A -85,B 0,C 180,E1 -12686.713,E2 -12686.713} C_VEL
LIN {X 0,Y 367.803,Z 850.569,A -85,B 0,C 180,E1 -12687.81,E2 -12687.81} C_VEL
LIN {X 0,Y 367.838,Z 851.181,A -85,B 0,C 180,E1 -12688.905,E2 -12688.905} C_VEL
LIN {X 0,Y 367.819,Z 851.337,A -85,B 0,C 180,E1 -12690,E2 -12690} C_VEL
LIN {X 0,Y 367.857,Z 851.091,A -85,B 0,C 180,E1 -12691.095,E2 -12691.095} C_VEL
LIN {X 0,Y 367.825,Z 850.434,A -85,B 0,C 180,E1 -12692.19,E2 -12692.19} C_VEL
LIN {X 0,Y 367.766,Z 849.349,A -85,B 0,C 180,E1 -12693.286,E2 -12693.286} C_VEL
LIN {X 0,Y 367.64,Z 847.787,A -85,B 0,C 180,E1 -12694.385,E2 -12694.385} C_VEL
LIN {X 0,Y 367.715,Z 843.909,A -85,B 0,C 180,E1 -12696.353,E2 -12696.353} C_VEL
LIN {X 0,Y 367.823,Z 838.721,A -85,B 0,C 180,E1 -12698.239,E2 -12698.239} C_VEL
LIN {X 0,Y 368.183,Z 832.289,A -85,B 0,C 180,E1 -12700.17,E2 -12700.17} C_VEL
LIN {X 0,Y 368.83,Z 825.346,A -85,B 0,C 180,E1 -12701.82,E2 -12701.82} C_VEL
LIN {X 0,Y 369.668,Z 816.675,A -85,B 0,C 180,E1 -12703.467,E2 -12703.467} C_VEL
LIN {X 0,Y 370.617,Z 806.957,A -85,B 0,C 180,E1 -12704.953,E2 -12704.953} C_VEL
LIN {X 0,Y 371.763,Z 796.876,A -85,B 0,C 180,E1 -12706.191,E2 -12706.191} C_VEL
LIN {X 0,Y 372.972,Z 785.836,A -85,B 0,C 180,E1 -12707.264,E2 -12707.264} C_VEL
LIN {X 0,Y 374.073,Z 773.49,A -85,B 0,C 180,E1 -12708.2,E2 -12708.2} C_VEL
LIN {X 0,Y 375.12,Z 760.95,A -85,B 0,C 180,E1 -12708.891,E2 -12708.891} C_VEL
LIN {X 0,Y 375.872,Z 747.69,A -85,B 0,C 180,E1 -12709.383,E2 -12709.383} C_VEL
LIN {X 0,Y 376.439,Z 720.577,A -85,B 0,C 180,E1 -12709.949,E2 -12709.949} C_VEL
LIN {X 0,Y 377.066,Z 672.702,A -85,B 0,C 180,E1 -12710.89,E2 -12710.89} C_VEL
LIN {X 0,Y 373.436,Z 641.809,A -85,B 0,C 180,E1 -12711.777,E2 -12711.777} C_VEL
LIN {X 0,Y 372.152,Z 632.398,A -85,B 0,C 180,E1 -12712.095,E2 -12712.095} C_VEL
LIN {X 0,Y 374.134,Z 609.729,A -85,B 0,C 180,E1 -12715.896,E2 -12715.896} C_VEL
LIN {X 0,Y 373.899,Z 606.259,A -85,B 0,C 180,E1 -12716.513,E2 -12716.513} C_VEL
LIN {X 0,Y 370.937,Z 592.938,A -85,B 0,C 180,E1 -12719.045,E2 -12719.045} C_VEL
LIN {X 0,Y 368.93,Z 584.531,A -85,B 0,C 180,E1 -12720.714,E2 -12720.714} C_VEL
LIN {X 0,Y 368.897,Z 584.535,A -85,B 0,C 180,E1 -12723.537,E2 -12723.537} C_VEL
LIN {X 0,Y 368.901,Z 584.532,A -85,B 0,C 180,E1 -12726.855,E2 -12726.855} C_VEL
LIN {X 0,Y 368.95,Z 584.527,A -85,B 0,C 180,E1 -12730.364,E2 -12730.364} C_VEL
LIN {X 0,Y 368.897,Z 584.533,A -85,B 0,C 180,E1 -12733.618,E2 -12733.618} C_VEL
LIN {X 0,Y 368.937,Z 584.527,A -85,B 0,C 180,E1 -12736.703,E2 -12736.703} C_VEL
LIN {X 0,Y 368.948,Z 584.522,A -85,B 0,C 180,E1 -12739.635,E2 -12739.635} C_VEL
LIN {X 0,Y 368.898,Z 584.531,A -85,B 0,C 180,E1 -12743.143,E2 -12743.143} C_VEL
LIN {X 0,Y 368.894,Z 584.527,A -85,B 0,C 180,E1 -12746.461,E2 -12746.461} C_VEL
LIN {X 0,Y 368.917,Z 584.52,A -85,B 0,C 180,E1 -12750.31,E2 -12750.31} C_VEL
LIN {X 0,Y 368.975,Z 584.521,A -85,B 0,C 180,E1 -12753.535,E2 -12753.535} C_VEL
LIN {X 0,Y 368.959,Z 584.513,A -85,B 0,C 180,E1 -12756.421,E2 -12756.421} C_VEL
LIN {X 0,Y 368.929,Z 584.526,A -85,B 0,C 180,E1 -12759.947,E2 -12759.947} C_VEL
LIN {X 0,Y 368.967,Z 584.51,A -85,B 0,C 180,E1 -12763.398,E2 -12763.398} C_VEL
LIN {X 0,Y 369.049,Z 584.516,A -85,B 0,C 180,E1 -12766.79,E2 -12766.79} C_VEL
LIN {X 0,Y 369.059,Z 584.502,A -85,B 0,C 180,E1 -12770.131,E2 -12770.131} C_VEL
LIN {X 0,Y 369.198,Z 584.492,A -85,B 0,C 180,E1 -12773.442,E2 -12773.442} C_VEL
LIN {X 0,Y 369.311,Z 584.467,A -85,B 0,C 180,E1 -12777.819,E2 -12777.819} C_VEL
LIN {X 0,Y 369.451,Z 584.454,A -85,B 0,C 180,E1 -12780,E2 -12780} C_VEL
LIN {X 0,Y 369.31,Z 584.481,A -85,B 0,C 180,E1 -12782.181,E2 -12782.181} C_VEL
LIN {X 0,Y 369.191,Z 584.481,A -85,B 0,C 180,E1 -12786.58,E2 -12786.58} C_VEL
LIN {X 0,Y 369.113,Z 584.508,A -85,B 0,C 180,E1 -12788.762,E2 -12788.762} C_VEL
LIN {X 0,Y 368.997,Z 584.507,A -85,B 0,C 180,E1 -12792.094,E2 -12792.094} C_VEL
LIN {X 0,Y 368.989,Z 584.521,A -85,B 0,C 180,E1 -12795.465,E2 -12795.465} C_VEL
LIN {X 0,Y 368.959,Z 584.513,A -85,B 0,C 180,E1 -12798.894,E2 -12798.894} C_VEL
LIN {X 0,Y 368.915,Z 584.53,A -85,B 0,C 180,E1 -12802.396,E2 -12802.396} C_VEL
LIN {X 0,Y 368.993,Z 584.516,A -85,B 0,C 180,E1 -12805.981,E2 -12805.981} C_VEL
LIN {X 0,Y 368.961,Z 584.522,A -85,B 0,C 180,E1 -12808.814,E2 -12808.814} C_VEL
LIN {X 0,Y 368.904,Z 584.531,A -85,B 0,C 180,E1 -12812.238,E2 -12812.238} C_VEL
LIN {X 0,Y 368.924,Z 584.523,A -85,B 0,C 180,E1 -12815.002,E2 -12815.002} C_VEL
LIN {X 0,Y 368.907,Z 584.531,A -85,B 0,C 180,E1 -12818.642,E2 -12818.642} C_VEL
LIN {X 0,Y 368.905,Z 584.506,A -85,B 0,C 180,E1 -12821.82,E2 -12821.82} C_VEL
LIN {X 0,Y 368.923,Z 584.533,A -85,B 0,C 180,E1 -12825.184,E2 -12825.184} C_VEL
LIN {X 0,Y 368.879,Z 584.521,A -85,B 0,C 180,E1 -12828.178,E2 -12828.178} C_VEL
LIN {X 0,Y 368.907,Z 584.523,A -85,B 0,C 180,E1 -12831.36,E2 -12831.36} C_VEL
LIN {X 0,Y 368.935,Z 584.53,A -85,B 0,C 180,E1 -12835.147,E2 -12835.147} C_VEL
LIN {X 0,Y 368.94,Z 584.529,A -85,B 0,C 180,E1 -12835.631,E2 -12835.631} C_VEL
LIN {X 0,Y 370.015,Z 587.532,A -85,B 0,C 180,E1 -12835.798,E2 -12835.798} C_VEL
LIN {X 0,Y 378.48,Z 605.826,A -85,B 0,C 180,E1 -12836.8,E2 -12836.8} C_VEL
LIN {X 0,Y 378.824,Z 606.681,A -85,B 0,C 180,E1 -12836.842,E2 -12836.842} C_VEL
LIN {X 0,Y 377.354,Z 683.305,A -85,B 0,C 180,E1 -12838.329,E2 -12838.329} C_VEL
LIN {X 0,Y 376.999,Z 696.688,A -85,B 0,C 180,E1 -12838.79,E2 -12838.79} C_VEL
LIN {X 0,Y 376.449,Z 708.919,A -85,B 0,C 180,E1 -12839.429,E2 -12839.429} C_VEL
LIN {X 0,Y 375.595,Z 720.856,A -85,B 0,C 180,E1 -12840.274,E2 -12840.274} C_VEL
LIN {X 0,Y 374.618,Z 731.754,A -85,B 0,C 180,E1 -12841.267,E2 -12841.267} C_VEL
LIN {X 0,Y 373.581,Z 741.818,A -85,B 0,C 180,E1 -12842.416,E2 -12842.416} C_VEL
LIN {X 0,Y 372.562,Z 750.809,A -85,B 0,C 180,E1 -12843.686,E2 -12843.686} C_VEL
LIN {X 0,Y 371.485,Z 759.741,A -85,B 0,C 180,E1 -12845.244,E2 -12845.244} C_VEL
LIN {X 0,Y 370.549,Z 767.061,A -85,B 0,C 180,E1 -12846.825,E2 -12846.825} C_VEL
LIN {X 0,Y 369.816,Z 772.616,A -85,B 0,C 180,E1 -12848.308,E2 -12848.308} C_VEL
LIN {X 0,Y 369.133,Z 777.574,A -85,B 0,C 180,E1 -12849.959,E2 -12849.959} C_VEL
LIN {X 0,Y 368.639,Z 781.483,A -85,B 0,C 180,E1 -12851.666,E2 -12851.666} C_VEL
LIN {X 0,Y 368.262,Z 784.301,A -85,B 0,C 180,E1 -12853.366,E2 -12853.366} C_VEL
LIN {X 0,Y 368.034,Z 785.608,A -85,B 0,C 180,E1 -12854.494,E2 -12854.494} C_VEL
LIN {X 0,Y 367.915,Z 786.509,A -85,B 0,C 180,E1 -12855.622,E2 -12855.622} C_VEL
LIN {X 0,Y 367.827,Z 787.031,A -85,B 0,C 180,E1 -12857.021,E2 -12857.021} C_VEL
LIN {X 0,Y 367.769,Z 786.705,A -85,B 0,C 180,E1 -12858.983,E2 -12858.983} C_VEL
LIN {X 0,Y 367.808,Z 785.979,A -85,B 0,C 180,E1 -12860.098,E2 -12860.098} C_VEL
LIN {X 0,Y 367.895,Z 784.808,A -85,B 0,C 180,E1 -12861.209,E2 -12861.209} C_VEL
LIN {X 0,Y 368.16,Z 781.942,A -85,B 0,C 180,E1 -12863.053,E2 -12863.053} C_VEL
LIN {X 0,Y 368.519,Z 777.376,A -85,B 0,C 180,E1 -12865.077,E2 -12865.077} C_VEL
LIN {X 0,Y 368.886,Z 772.395,A -85,B 0,C 180,E1 -12866.724,E2 -12866.724} C_VEL
LIN {X 0,Y 369.51,Z 766.085,A -85,B 0,C 180,E1 -12868.365,E2 -12868.365} C_VEL
LIN {X 0,Y 370.187,Z 758.26,A -85,B 0,C 180,E1 -12870,E2 -12870} C_VEL
LIN {X 0,Y 371.002,Z 750.25,A -85,B 0,C 180,E1 -12871.357,E2 -12871.357} C_VEL
LIN {X 0,Y 371.827,Z 740.499,A -85,B 0,C 180,E1 -12872.708,E2 -12872.708} C_VEL
LIN {X 0,Y 372.69,Z 729.536,A -85,B 0,C 180,E1 -12873.92,E2 -12873.92} C_VEL
LIN {X 0,Y 373.496,Z 718.831,A -85,B 0,C 180,E1 -12874.857,E2 -12874.857} C_VEL
LIN {X 0,Y 374.146,Z 707.048,A -85,B 0,C 180,E1 -12875.659,E2 -12875.659} C_VEL
LIN {X 0,Y 374.6,Z 694.182,A -85,B 0,C 180,E1 -12876.294,E2 -12876.294} C_VEL
LIN {X 0,Y 374.945,Z 681.778,A -85,B 0,C 180,E1 -12876.694,E2 -12876.694} C_VEL
LIN {X 0,Y 376.002,Z 603.348,A -85,B 0,C 180,E1 -12878.2,E2 -12878.2} C_VEL
LIN {X 0,Y 374.627,Z 599.609,A -85,B 0,C 180,E1 -12878.341,E2 -12878.341} C_VEL
LIN {X 0,Y 373.192,Z 597.697,A -85,B 0,C 180,E1 -12878.449,E2 -12878.449} C_VEL
LIN {X 0,Y 365.942,Z 593.804,A -85,B 0,C 180,E1 -12878.892,E2 -12878.892} C_VEL
LIN {X 0,Y 364.432,Z 591.924,A -85,B 0,C 180,E1 -12879.007,E2 -12879.007} C_VEL
LIN {X 0,Y 362.042,Z 585.387,A -85,B 0,C 180,E1 -12879.278,E2 -12879.278} C_VEL
LIN {X 0,Y 362.002,Z 585.39,A -85,B 0,C 180,E1 -12883.472,E2 -12883.472} C_VEL
LIN {X 0,Y 361.935,Z 585.399,A -85,B 0,C 180,E1 -12886.933,E2 -12886.933} C_VEL
LIN {X 0,Y 361.888,Z 585.404,A -85,B 0,C 180,E1 -12890.46,E2 -12890.46} C_VEL
LIN {X 0,Y 361.912,Z 585.403,A -85,B 0,C 180,E1 -12894.425,E2 -12894.425} C_VEL
LIN {X 0,Y 365.944,Z 596.001,A -85,B 0,C 180,E1 -12894.898,E2 -12894.898} C_VEL
LIN {X 0,Y 369.878,Z 606.567,A -85,B 0,C 180,E1 -12895.347,E2 -12895.347} C_VEL
LIN {X 0,Y 368.337,Z 683.916,A -85,B 0,C 180,E1 -12896.97,E2 -12896.97} C_VEL
LIN {X 0,Y 367.963,Z 697.451,A -85,B 0,C 180,E1 -12897.475,E2 -12897.475} C_VEL
LIN {X 0,Y 367.465,Z 708.911,A -85,B 0,C 180,E1 -12898.096,E2 -12898.096} C_VEL
LIN {X 0,Y 366.73,Z 720.668,A -85,B 0,C 180,E1 -12898.939,E2 -12898.939} C_VEL
LIN {X 0,Y 365.95,Z 731.618,A -85,B 0,C 180,E1 -12899.954,E2 -12899.954} C_VEL
LIN {X 0,Y 365.036,Z 742.135,A -85,B 0,C 180,E1 -12901.172,E2 -12901.172} C_VEL
LIN {X 0,Y 364.173,Z 751.486,A -85,B 0,C 180,E1 -12902.505,E2 -12902.505} C_VEL
LIN {X 0,Y 363.467,Z 758.711,A -85,B 0,C 180,E1 -12903.752,E2 -12903.752} C_VEL
LIN {X 0,Y 362.579,Z 767.248,A -85,B 0,C 180,E1 -12905.555,E2 -12905.555} C_VEL
LIN {X 0,Y 362.029,Z 773.589,A -85,B 0,C 180,E1 -12907.257,E2 -12907.257} C_VEL
LIN {X 0,Y 361.541,Z 778.623,A -85,B 0,C 180,E1 -12908.962,E2 -12908.962} C_VEL
LIN {X 0,Y 361.171,Z 782.414,A -85,B 0,C 180,E1 -12910.633,E2 -12910.633} C_VEL
LIN {X 0,Y 360.897,Z 785.139,A -85,B 0,C 180,E1 -12912.268,E2 -12912.268} C_VEL
LIN {X 0,Y 360.678,Z 787.451,A -85,B 0,C 180,E1 -12914.544,E2 -12914.544} C_VEL
LIN {X 0,Y 360.667,Z 788.033,A -85,B 0,C 180,E1 -12916.134,E2 -12916.134} C_VEL
LIN {X 0,Y 360.746,Z 787.795,A -85,B 0,C 180,E1 -12917.756,E2 -12917.756} C_VEL
LIN {X 0,Y 361.033,Z 786.055,A -85,B 0,C 180,E1 -12920.03,E2 -12920.03} C_VEL
LIN {X 0,Y 361.535,Z 782.729,A -85,B 0,C 180,E1 -12922.214,E2 -12922.214} C_VEL
LIN {X 0,Y 362.111,Z 777.697,A -85,B 0,C 180,E1 -12924.391,E2 -12924.391} C_VEL
LIN {X 0,Y 362.9,Z 771.375,A -85,B 0,C 180,E1 -12926.38,E2 -12926.38} C_VEL
LIN {X 0,Y 363.626,Z 765.824,A -85,B 0,C 180,E1 -12927.757,E2 -12927.757} C_VEL
LIN {X 0,Y 364.548,Z 758.4,A -85,B 0,C 180,E1 -12929.277,E2 -12929.277} C_VEL
LIN {X 0,Y 365.635,Z 749.125,A -85,B 0,C 180,E1 -12930.808,E2 -12930.808} C_VEL
LIN {X 0,Y 366.749,Z 739.017,A -85,B 0,C 180,E1 -12932.143,E2 -12932.143} C_VEL
LIN {X 0,Y 367.756,Z 728.19,A -85,B 0,C 180,E1 -12933.294,E2 -12933.294} C_VEL
LIN {X 0,Y 368.59,Z 717.156,A -85,B 0,C 180,E1 -12934.216,E2 -12934.216} C_VEL
LIN {X 0,Y 369.346,Z 704.362,A -85,B 0,C 180,E1 -12935.027,E2 -12935.027} C_VEL
LIN {X 0,Y 369.807,Z 691.594,A -85,B 0,C 180,E1 -12935.607,E2 -12935.607} C_VEL
LIN {X 0,Y 370.104,Z 677.051,A -85,B 0,C 180,E1 -12936.002,E2 -12936.002} C_VEL
LIN {X 0,Y 371.694,Z 607.509,A -85,B 0,C 180,E1 -12937.495,E2 -12937.495} C_VEL
LIN {X 0,Y 364.386,Z 591.275,A -85,B 0,C 180,E1 -12938.428,E2 -12938.428} C_VEL
LIN {X 0,Y 361.991,Z 586.071,A -85,B 0,C 180,E1 -12938.748,E2 -12938.748} C_VEL
LIN {X 0,Y 361.872,Z 585.41,A -85,B 0,C 180,E1 -12938.78,E2 -12938.78} C_VEL
LIN {X 0,Y 361.96,Z 585.398,A -85,B 0,C 180,E1 -12942.061,E2 -12942.061} C_VEL
LIN {X 0,Y 361.99,Z 585.396,A -85,B 0,C 180,E1 -12946.101,E2 -12946.101} C_VEL
LIN {X 0,Y 362.028,Z 585.39,A -85,B 0,C 180,E1 -12949.938,E2 -12949.938} C_VEL
LIN {X 0,Y 362.143,Z 585.375,A -85,B 0,C 180,E1 -12952.192,E2 -12952.192} C_VEL
LIN {X 0,Y 362.116,Z 585.379,A -85,B 0,C 180,E1 -12954.431,E2 -12954.431} C_VEL
LIN {X 0,Y 362.275,Z 585.354,A -85,B 0,C 180,E1 -12957.776,E2 -12957.776} C_VEL
LIN {X 0,Y 362.421,Z 585.34,A -85,B 0,C 180,E1 -12960,E2 -12960} C_VEL
LIN {X 0,Y 362.275,Z 585.36,A -85,B 0,C 180,E1 -12962.224,E2 -12962.224} C_VEL
LIN {X 0,Y 362.161,Z 585.367,A -85,B 0,C 180,E1 -12966.686,E2 -12966.686} C_VEL
LIN {X 0,Y 362.028,Z 585.381,A -85,B 0,C 180,E1 -12970.062,E2 -12970.062} C_VEL
LIN {X 0,Y 361.99,Z 585.382,A -85,B 0,C 180,E1 -12973.899,E2 -12973.899} C_VEL
LIN {X 0,Y 361.96,Z 585.389,A -85,B 0,C 180,E1 -12977.939,E2 -12977.939} C_VEL
LIN {X 0,Y 361.885,Z 585.402,A -85,B 0,C 180,E1 -12981.653,E2 -12981.653} C_VEL
LIN {X 0,Y 361.921,Z 585.401,A -85,B 0,C 180,E1 -12985.291,E2 -12985.291} C_VEL
LIN {X 0,Y 361.916,Z 585.396,A -85,B 0,C 180,E1 -12987.778,E2 -12987.778} C_VEL
LIN {X 0,Y 361.842,Z 585.41,A -85,B 0,C 180,E1 -12991.286,E2 -12991.286} C_VEL
LIN {X 0,Y 361.849,Z 585.408,A -85,B 0,C 180,E1 -12994.281,E2 -12994.281} C_VEL
LIN {X 0,Y 361.861,Z 585.409,A -85,B 0,C 180,E1 -12997.224,E2 -12997.224} C_VEL
LIN {X 0,Y 361.901,Z 585.405,A -85,B 0,C 180,E1 -13000.769,E2 -13000.769} C_VEL
LIN {X 0,Y 361.9,Z 585.406,A -85,B 0,C 180,E1 -13004.356,E2 -13004.356} C_VEL
LIN {X 0,Y 361.854,Z 585.411,A -85,B 0,C 180,E1 -13007.565,E2 -13007.565} C_VEL
LIN {X 0,Y 361.872,Z 585.409,A -85,B 0,C 180,E1 -13010.973,E2 -13010.973} C_VEL
LIN {X 0,Y 361.873,Z 585.409,A -85,B 0,C 180,E1 -13014.656,E2 -13014.656} C_VEL
LIN {X 0,Y 361.865,Z 585.428,A -85,B 0,C 180,E1 -13016.548,E2 -13016.548} C_VEL
LIN {X 0,Y 364.861,Z 597.692,A -85,B 0,C 180,E1 -13019.628,E2 -13019.628} C_VEL
LIN {X 0,Y 367.13,Z 609.398,A -85,B 0,C 180,E1 -13022.354,E2 -13022.354} C_VEL
LIN {X 0,Y 366.197,Z 619.47,A -85,B 0,C 180,E1 -13024.425,E2 -13024.425} C_VEL
LIN {X 0,Y 364.722,Z 634.15,A -85,B 0,C 180,E1 -13027.355,E2 -13027.355} C_VEL
LIN {X 0,Y 367.876,Z 653.996,A -85,B 0,C 180,E1 -13028.052,E2 -13028.052} C_VEL
LIN {X 0,Y 370.525,Z 676.56,A -85,B 0,C 180,E1 -13028.759,E2 -13028.759} C_VEL
LIN {X 0,Y 369.155,Z 745.211,A -85,B 0,C 180,E1 -13030.25,E2 -13030.25} C_VEL
LIN {X 0,Y 368.34,Z 758.676,A -85,B 0,C 180,E1 -13030.748,E2 -13030.748} C_VEL
LIN {X 0,Y 367.293,Z 771.571,A -85,B 0,C 180,E1 -13031.452,E2 -13031.452} C_VEL
LIN {X 0,Y 366.235,Z 782.625,A -85,B 0,C 180,E1 -13032.264,E2 -13032.264} C_VEL
LIN {X 0,Y 365.013,Z 794.254,A -85,B 0,C 180,E1 -13033.358,E2 -13033.358} C_VEL
LIN {X 0,Y 363.896,Z 804.94,A -85,B 0,C 180,E1 -13034.619,E2 -13034.619} C_VEL
LIN {X 0,Y 362.989,Z 814.333,A -85,B 0,C 180,E1 -13035.995,E2 -13035.995} C_VEL
LIN {X 0,Y 362.094,Z 822.201,A -85,B 0,C 180,E1 -13037.388,E2 -13037.388} C_VEL
LIN {X 0,Y 361.301,Z 829.951,A -85,B 0,C 180,E1 -13039.068,E2 -13039.068} C_VEL
LIN {X 0,Y 360.942,Z 835.283,A -85,B 0,C 180,E1 -13040.474,E2 -13040.474} C_VEL
LIN {X 0,Y 360.696,Z 840.48,A -85,B 0,C 180,E1 -13042.161,E2 -13042.161} C_VEL
LIN {X 0,Y 360.587,Z 844.286,A -85,B 0,C 180,E1 -13043.729,E2 -13043.729} C_VEL
LIN {X 0,Y 360.554,Z 847.509,A -85,B 0,C 180,E1 -13045.528,E2 -13045.528} C_VEL
LIN {X 0,Y 360.634,Z 848.944,A -85,B 0,C 180,E1 -13046.648,E2 -13046.648} C_VEL
LIN {X 0,Y 360.733,Z 849.971,A -85,B 0,C 180,E1 -13047.767,E2 -13047.767} C_VEL
LIN {X 0,Y 360.774,Z 850.566,A -85,B 0,C 180,E1 -13048.884,E2 -13048.884} C_VEL
LIN {X 0,Y 360.772,Z 850.711,A -85,B 0,C 180,E1 -13050,E2 -13050} C_VEL
LIN {X 0,Y 360.809,Z 850.454,A -85,B 0,C 180,E1 -13051.116,E2 -13051.116} C_VEL
LIN {X 0,Y 360.754,Z 849.786,A -85,B 0,C 180,E1 -13052.233,E2 -13052.233} C_VEL
LIN {X 0,Y 360.688,Z 848.676,A -85,B 0,C 180,E1 -13053.351,E2 -13053.351} C_VEL
LIN {X 0,Y 360.567,Z 847.099,A -85,B 0,C 180,E1 -13054.472,E2 -13054.472} C_VEL
LIN {X 0,Y 360.627,Z 843.527,A -85,B 0,C 180,E1 -13056.329,E2 -13056.329} C_VEL
LIN {X 0,Y 360.828,Z 836.603,A -85,B 0,C 180,E1 -13058.964,E2 -13058.964} C_VEL
LIN {X 0,Y 361.295,Z 829.749,A -85,B 0,C 180,E1 -13060.933,E2 -13060.933} C_VEL
LIN {X 0,Y 362.107,Z 822.325,A -85,B 0,C 180,E1 -13062.612,E2 -13062.612} C_VEL
LIN {X 0,Y 362.953,Z 814.784,A -85,B 0,C 180,E1 -13064.007,E2 -13064.007} C_VEL
LIN {X 0,Y 363.864,Z 805.663,A -85,B 0,C 180,E1 -13065.401,E2 -13065.401} C_VEL
LIN {X 0,Y 365.065,Z 795.564,A -85,B 0,C 180,E1 -13066.64,E2 -13066.64} C_VEL
LIN {X 0,Y 366.402,Z 784.368,A -85,B 0,C 180,E1 -13067.728,E2 -13067.728} C_VEL
LIN {X 0,Y 367.345,Z 773.778,A -85,B 0,C 180,E1 -13068.546,E2 -13068.546} C_VEL
LIN {X 0,Y 368.501,Z 760.963,A -85,B 0,C 180,E1 -13069.279,E2 -13069.279} C_VEL
LIN {X 0,Y 369.293,Z 748.015,A -85,B 0,C 180,E1 -13069.779,E2 -13069.779} C_VEL
LIN {X 0,Y 369.704,Z 729.445,A -85,B 0,C 180,E1 -13070.199,E2 -13070.199} C_VEL
LIN {X 0,Y 370.613,Z 673.875,A -85,B 0,C 180,E1 -13071.302,E2 -13071.302} C_VEL
LIN {X 0,Y 367.149,Z 644.09,A -85,B 0,C 180,E1 -13072.179,E2 -13072.179} C_VEL
LIN {X 0,Y 365.297,Z 630.982,A -85,B 0,C 180,E1 -13072.63,E2 -13072.63} C_VEL
LIN {X 0,Y 367.222,Z 610.605,A -85,B 0,C 180,E1 -13076.115,E2 -13076.115} C_VEL
LIN {X 0,Y 366.507,Z 605.349,A -85,B 0,C 180,E1 -13077.091,E2 -13077.091} C_VEL
LIN {X 0,Y 363.063,Z 590.414,A -85,B 0,C 180,E1 -13080.012,E2 -13080.012} C_VEL
LIN {X 0,Y 361.885,Z 585.408,A -85,B 0,C 180,E1 -13081.06,E2 -13081.06} C_VEL
LIN {X 0,Y 361.854,Z 585.413,A -85,B 0,C 180,E1 -13084.279,E2 -13084.279} C_VEL
LIN {X 0,Y 361.87,Z 585.408,A -85,B 0,C 180,E1 -13087.224,E2 -13087.224} C_VEL
LIN {X 0,Y 361.87,Z 585.406,A -85,B 0,C 180,E1 -13090.761,E2 -13090.761} C_VEL
LIN {X 0,Y 361.862,Z 585.408,A -85,B 0,C 180,E1 -13094.36,E2 -13094.36} C_VEL
LIN {X 0,Y 361.88,Z 585.405,A -85,B 0,C 180,E1 -13097.559,E2 -13097.559} C_VEL
LIN {X 0,Y 361.87,Z 585.402,A -85,B 0,C 180,E1 -13100.972,E2 -13100.972} C_VEL
LIN {X 0,Y 361.869,Z 585.397,A -85,B 0,C 180,E1 -13104.654,E2 -13104.654} C_VEL
LIN {X 0,Y 361.853,Z 585.412,A -85,B 0,C 180,E1 -13108.372,E2 -13108.372} C_VEL
LIN {X 0,Y 361.916,Z 585.393,A -85,B 0,C 180,E1 -13112.221,E2 -13112.221} C_VEL
LIN {X 0,Y 361.921,Z 585.401,A -85,B 0,C 180,E1 -13114.709,E2 -13114.709} C_VEL
LIN {X 0,Y 361.884,Z 585.394,A -85,B 0,C 180,E1 -13118.347,E2 -13118.347} C_VEL
LIN {X 0,Y 361.96,Z 585.396,A -85,B 0,C 180,E1 -13122.061,E2 -13122.061} C_VEL
LIN {X 0,Y 361.99,Z 585.387,A -85,B 0,C 180,E1 -13126.101,E2 -13126.101} C_VEL
LIN {X 0,Y 362.023,Z 585.381,A -85,B 0,C 180,E1 -13129.938,E2 -13129.938} C_VEL
LIN {X 0,Y 362.159,Z 585.369,A -85,B 0,C 180,E1 -13133.314,E2 -13133.314} C_VEL
LIN {X 0,Y 362.275,Z 585.343,A -85,B 0,C 180,E1 -13137.776,E2 -13137.776} C_VEL
LIN {X 0,Y 362.421,Z 585.33,A -85,B 0,C 180,E1 -13140,E2 -13140} C_VEL
LIN {X 0,Y 362.274,Z 585.357,A -85,B 0,C 180,E1 -13142.224,E2 -13142.224} C_VEL
LIN {X 0,Y 362.155,Z 585.358,A -85,B 0,C 180,E1 -13146.686,E2 -13146.686} C_VEL
LIN {X 0,Y 362.023,Z 585.387,A -85,B 0,C 180,E1 -13150.062,E2 -13150.062} C_VEL
LIN {X 0,Y 361.99,Z 585.386,A -85,B 0,C 180,E1 -13153.899,E2 -13153.899} C_VEL
LIN {X 0,Y 361.96,Z 585.388,A -85,B 0,C 180,E1 -13157.939,E2 -13157.939} C_VEL
LIN {X 0,Y 361.881,Z 585.406,A -85,B 0,C 180,E1 -13161.654,E2 -13161.654} C_VEL
LIN {X 0,Y 361.92,Z 585.394,A -85,B 0,C 180,E1 -13165.291,E2 -13165.291} C_VEL
LIN {X 0,Y 361.916,Z 585.401,A -85,B 0,C 180,E1 -13167.778,E2 -13167.778} C_VEL
LIN {X 0,Y 361.854,Z 585.411,A -85,B 0,C 180,E1 -13171.628,E2 -13171.628} C_VEL
LIN {X 0,Y 361.869,Z 585.406,A -85,B 0,C 180,E1 -13175.346,E2 -13175.346} C_VEL
LIN {X 0,Y 361.869,Z 585.411,A -85,B 0,C 180,E1 -13179.028,E2 -13179.028} C_VEL
LIN {X 0,Y 361.852,Z 585.384,A -85,B 0,C 180,E1 -13182.436,E2 -13182.436} C_VEL
LIN {X 0,Y 361.832,Z 585.41,A -85,B 0,C 180,E1 -13185.945,E2 -13185.945} C_VEL
LIN {X 0,Y 361.832,Z 585.408,A -85,B 0,C 180,E1 -13189.245,E2 -13189.245} C_VEL
LIN {X 0,Y 361.863,Z 585.401,A -85,B 0,C 180,E1 -13192.778,E2 -13192.778} C_VEL
LIN {X 0,Y 361.903,Z 585.405,A -85,B 0,C 180,E1 -13195.104,E2 -13195.104} C_VEL
LIN {X 0,Y 362.952,Z 588.35,A -85,B 0,C 180,E1 -13195.268,E2 -13195.268} C_VEL
LIN {X 0,Y 371.428,Z 606.328,A -85,B 0,C 180,E1 -13196.302,E2 -13196.302} C_VEL
LIN {X 0,Y 372.39,Z 609.116,A -85,B 0,C 180,E1 -13196.431,E2 -13196.431} C_VEL
LIN {X 0,Y 370.847,Z 683.609,A -85,B 0,C 180,E1 -13197.897,E2 -13197.897} C_VEL
LIN {X 0,Y 370.48,Z 696.993,A -85,B 0,C 180,E1 -13198.362,E2 -13198.362} C_VEL
LIN {X 0,Y 369.919,Z 709.273,A -85,B 0,C 180,E1 -13199.008,E2 -13199.008} C_VEL
LIN {X 0,Y 369.028,Z 721.035,A -85,B 0,C 180,E1 -13199.848,E2 -13199.848} C_VEL
LIN {X 0,Y 367.997,Z 732.007,A -85,B 0,C 180,E1 -13200.857,E2 -13200.857} C_VEL
LIN {X 0,Y 366.8,Z 743.044,A -85,B 0,C 180,E1 -13202.144,E2 -13202.144} C_VEL
LIN {X 0,Y 365.724,Z 752.09,A -85,B 0,C 180,E1 -13203.463,E2 -13203.463} C_VEL
LIN {X 0,Y 364.578,Z 761.19,A -85,B 0,C 180,E1 -13205.105,E2 -13205.105} C_VEL
LIN {X 0,Y 363.431,Z 769.228,A -85,B 0,C 180,E1 -13206.947,E2 -13206.947} C_VEL
LIN {X 0,Y 362.701,Z 774.465,A -85,B 0,C 180,E1 -13208.449,E2 -13208.449} C_VEL
LIN {X 0,Y 362.048,Z 779.159,A -85,B 0,C 180,E1 -13210.142,E2 -13210.142} C_VEL
LIN {X 0,Y 361.534,Z 782.814,A -85,B 0,C 180,E1 -13211.879,E2 -13211.879} C_VEL
LIN {X 0,Y 361.291,Z 784.67,A -85,B 0,C 180,E1 -13213.035,E2 -13213.035} C_VEL
LIN {X 0,Y 361.02,Z 786.046,A -85,B 0,C 180,E1 -13214.185,E2 -13214.185} C_VEL
LIN {X 0,Y 360.877,Z 786.996,A -85,B 0,C 180,E1 -13215.335,E2 -13215.335} C_VEL
LIN {X 0,Y 360.781,Z 787.631,A -85,B 0,C 180,E1 -13216.907,E2 -13216.907} C_VEL
LIN {X 0,Y 360.712,Z 787.385,A -85,B 0,C 180,E1 -13218.765,E2 -13218.765} C_VEL
LIN {X 0,Y 360.727,Z 786.709,A -85,B 0,C 180,E1 -13219.901,E2 -13219.901} C_VEL
LIN {X 0,Y 360.798,Z 785.635,A -85,B 0,C 180,E1 -13221.035,E2 -13221.035} C_VEL
LIN {X 0,Y 361.089,Z 782.635,A -85,B 0,C 180,E1 -13223.041,E2 -13223.041} C_VEL
LIN {X 0,Y 361.434,Z 778.408,A -85,B 0,C 180,E1 -13224.98,E2 -13224.98} C_VEL
LIN {X 0,Y 361.803,Z 773.549,A -85,B 0,C 180,E1 -13226.659,E2 -13226.659} C_VEL
LIN {X 0,Y 362.442,Z 767.412,A -85,B 0,C 180,E1 -13228.333,E2 -13228.333} C_VEL
LIN {X 0,Y 363.126,Z 759.74,A -85,B 0,C 180,E1 -13230,E2 -13230} C_VEL
LIN {X 0,Y 364.103,Z 750.182,A -85,B 0,C 180,E1 -13231.659,E2 -13231.659} C_VEL
LIN {X 0,Y 364.954,Z 740.232,A -85,B 0,C 180,E1 -13233.036,E2 -13233.036} C_VEL
LIN {X 0,Y 365.89,Z 729.075,A -85,B 0,C 180,E1 -13234.268,E2 -13234.268} C_VEL
LIN {X 0,Y 366.731,Z 718.089,A -85,B 0,C 180,E1 -13235.223,E2 -13235.223} C_VEL
LIN {X 0,Y 367.376,Z 705.785,A -85,B 0,C 180,E1 -13236.039,E2 -13236.039} C_VEL
LIN {X 0,Y 367.855,Z 693.03,A -85,B 0,C 180,E1 -13236.651,E2 -13236.651} C_VEL
LIN {X 0,Y 368.16,Z 680.799,A -85,B 0,C 180,E1 -13237.024,E2 -13237.024} C_VEL
LIN {X 0,Y 369.179,Z 604.684,A -85,B 0,C 180,E1 -13238.508,E2 -13238.508} C_VEL
LIN {X 0,Y 364.432,Z 591.924,A -85,B 0,C 180,E1 -13239.007,E2 -13239.007} C_VEL
LIN {X 0,Y 363.264,Z 589.769,A -85,B 0,C 180,E1 -13239.189,E2 -13239.189} C_VEL
LIN {X 0,Y 361.559,Z 587.739,A -85,B 0,C 180,E1 -13239.59,E2 -13239.59} C_VEL
LIN {X 0,Y 359.493,Z 586.317,A -85,B 0,C 180,E1 -13240.243,E2 -13240.243} C_VEL
LIN {X 0,Y 357.735,Z 585.922,A -85,B 0,C 180,E1 -13240.988,E2 -13240.988} C_VEL
LIN {X 0,Y 355.777,Z 586.17,A -85,B 0,C 180,E1 -13242.194,E2 -13242.194} C_VEL
LIN {X 0,Y 354.982,Z 586.273,A -85,B 0,C 180,E1 -13243.256,E2 -13243.256} C_VEL
LIN {X 0,Y 354.943,Z 586.27,A -85,B 0,C 180,E1 -13243.613,E2 -13243.613} C_VEL
LIN {X 0,Y 354.9,Z 586.276,A -85,B 0,C 180,E1 -13247.28,E2 -13247.28} C_VEL
LIN {X 0,Y 354.827,Z 586.282,A -85,B 0,C 180,E1 -13250.886,E2 -13250.886} C_VEL
LIN {X 0,Y 354.868,Z 586.284,A -85,B 0,C 180,E1 -13254.043,E2 -13254.043} C_VEL
LIN {X 0,Y 363.053,Z 607.355,A -85,B 0,C 180,E1 -13254.994,E2 -13254.994} C_VEL
LIN {X 0,Y 361.547,Z 685.343,A -85,B 0,C 180,E1 -13256.682,E2 -13256.682} C_VEL
LIN {X 0,Y 361.153,Z 698.911,A -85,B 0,C 180,E1 -13257.212,E2 -13257.212} C_VEL
LIN {X 0,Y 360.555,Z 710.928,A -85,B 0,C 180,E1 -13257.892,E2 -13257.892} C_VEL
LIN {X 0,Y 359.73,Z 723.41,A -85,B 0,C 180,E1 -13258.849,E2 -13258.849} C_VEL
LIN {X 0,Y 358.895,Z 734.612,A -85,B 0,C 180,E1 -13259.956,E2 -13259.956} C_VEL
LIN {X 0,Y 357.981,Z 744.628,A -85,B 0,C 180,E1 -13261.184,E2 -13261.184} C_VEL
LIN {X 0,Y 357.123,Z 753.205,A -85,B 0,C 180,E1 -13262.471,E2 -13262.471} C_VEL
LIN {X 0,Y 356.255,Z 761.773,A -85,B 0,C 180,E1 -13264.049,E2 -13264.049} C_VEL
LIN {X 0,Y 355.406,Z 769.567,A -85,B 0,C 180,E1 -13265.83,E2 -13265.83} C_VEL
LIN {X 0,Y 354.871,Z 775.732,A -85,B 0,C 180,E1 -13267.611,E2 -13267.611} C_VEL
LIN {X 0,Y 354.361,Z 780.53,A -85,B 0,C 180,E1 -13269.393,E2 -13269.393} C_VEL
LIN {X 0,Y 354.032,Z 783.895,A -85,B 0,C 180,E1 -13271.031,E2 -13271.031} C_VEL
LIN {X 0,Y 353.767,Z 786.354,A -85,B 0,C 180,E1 -13272.688,E2 -13272.688} C_VEL
LIN {X 0,Y 353.612,Z 787.892,A -85,B 0,C 180,E1 -13274.316,E2 -13274.316} C_VEL
LIN {X 0,Y 353.59,Z 788.605,A -85,B 0,C 180,E1 -13275.92,E2 -13275.92} C_VEL
LIN {X 0,Y 353.679,Z 788.546,A -85,B 0,C 180,E1 -13277.498,E2 -13277.498} C_VEL
LIN {X 0,Y 353.804,Z 787.756,A -85,B 0,C 180,E1 -13279.041,E2 -13279.041} C_VEL
LIN {X 0,Y 354.282,Z 785.035,A -85,B 0,C 180,E1 -13281.398,E2 -13281.398} C_VEL
LIN {X 0,Y 354.837,Z 780.982,A -85,B 0,C 180,E1 -13283.545,E2 -13283.545} C_VEL
LIN {X 0,Y 355.523,Z 775.483,A -85,B 0,C 180,E1 -13285.586,E2 -13285.586} C_VEL
LIN {X 0,Y 356.484,Z 768.685,A -85,B 0,C 180,E1 -13287.505,E2 -13287.505} C_VEL
LIN {X 0,Y 357.522,Z 760.669,A -85,B 0,C 180,E1 -13289.263,E2 -13289.263} C_VEL
LIN {X 0,Y 358.709,Z 751.102,A -85,B 0,C 180,E1 -13290.936,E2 -13290.936} C_VEL
LIN {X 0,Y 359.94,Z 740.698,A -85,B 0,C 180,E1 -13292.372,E2 -13292.372} C_VEL
LIN {X 0,Y 361.01,Z 729.845,A -85,B 0,C 180,E1 -13293.571,E2 -13293.571} C_VEL
LIN {X 0,Y 361.932,Z 718.57,A -85,B 0,C 180,E1 -13294.556,E2 -13294.556} C_VEL
LIN {X 0,Y 362.748,Z 705.976,A -85,B 0,C 180,E1 -13295.383,E2 -13295.383} C_VEL
LIN {X 0,Y 363.22,Z 693.23,A -85,B 0,C 180,E1 -13295.99,E2 -13295.99} C_VEL
LIN {X 0,Y 363.557,Z 679.884,A -85,B 0,C 180,E1 -13296.381,E2 -13296.381} C_VEL
LIN {X 0,Y 365.254,Z 609.379,A -85,B 0,C 180,E1 -13297.926,E2 -13297.926} C_VEL
LIN {X 0,Y 358.443,Z 594.391,A -85,B 0,C 180,E1 -13298.83,E2 -13298.83} C_VEL
LIN {X 0,Y 354.938,Z 586.933,A -85,B 0,C 180,E1 -13299.31,E2 -13299.31} C_VEL
LIN {X 0,Y 354.835,Z 586.287,A -85,B 0,C 180,E1 -13299.341,E2 -13299.341} C_VEL
LIN {X 0,Y 354.891,Z 586.281,A -85,B 0,C 180,E1 -13302.719,E2 -13302.719} C_VEL
LIN {X 0,Y 354.944,Z 586.273,A -85,B 0,C 180,E1 -13306.255,E2 -13306.255} C_VEL
LIN {X 0,Y 354.975,Z 586.268,A -85,B 0,C 180,E1 -13309.736,E2 -13309.736} C_VEL
LIN {X 0,Y 355.106,Z 586.252,A -85,B 0,C 180,E1 -13312.037,E2 -13312.037} C_VEL
LIN {X 0,Y 355.089,Z 586.255,A -85,B 0,C 180,E1 -13314.321,E2 -13314.321} C_VEL
LIN {X 0,Y 355.238,Z 586.23,A -85,B 0,C 180,E1 -13317.732,E2 -13317.732} C_VEL
LIN {X 0,Y 355.39,Z 586.215,A -85,B 0,C 180,E1 -13320,E2 -13320} C_VEL
LIN {X 0,Y 355.238,Z 586.237,A -85,B 0,C 180,E1 -13322.268,E2 -13322.268} C_VEL
LIN {X 0,Y 355.124,Z 586.243,A -85,B 0,C 180,E1 -13326.82,E2 -13326.82} C_VEL
LIN {X 0,Y 354.974,Z 586.259,A -85,B 0,C 180,E1 -13330.264,E2 -13330.264} C_VEL
LIN {X 0,Y 354.935,Z 586.261,A -85,B 0,C 180,E1 -13334.019,E2 -13334.019} C_VEL
LIN {X 0,Y 354.916,Z 586.267,A -85,B 0,C 180,E1 -13338.109,E2 -13338.109} C_VEL
LIN {X 0,Y 354.828,Z 586.283,A -85,B 0,C 180,E1 -13342.107,E2 -13342.107} C_VEL
LIN {X 0,Y 354.893,Z 586.277,A -85,B 0,C 180,E1 -13345.828,E2 -13345.828} C_VEL
LIN {X 0,Y 354.848,Z 586.282,A -85,B 0,C 180,E1 -13349.679,E2 -13349.679} C_VEL
LIN {X 0,Y 354.801,Z 586.284,A -85,B 0,C 180,E1 -13353.703,E2 -13353.703} C_VEL
LIN {X 0,Y 354.794,Z 586.288,A -85,B 0,C 180,E1 -13356.46,E2 -13356.46} C_VEL
LIN {X 0,Y 354.82,Z 586.284,A -85,B 0,C 180,E1 -13359.424,E2 -13359.424} C_VEL
LIN {X 0,Y 354.83,Z 586.287,A -85,B 0,C 180,E1 -13362.876,E2 -13362.876} C_VEL
LIN {X 0,Y 354.801,Z 586.29,A -85,B 0,C 180,E1 -13366.11,E2 -13366.11} C_VEL
LIN {X 0,Y 354.822,Z 586.287,A -85,B 0,C 180,E1 -13369.185,E2 -13369.185} C_VEL
LIN {X 0,Y 354.807,Z 586.29,A -85,B 0,C 180,E1 -13372.403,E2 -13372.403} C_VEL
LIN {X 0,Y 354.807,Z 586.292,A -85,B 0,C 180,E1 -13376.022,E2 -13376.022} C_VEL
LIN {X 0,Y 357.587,Z 597.516,A -85,B 0,C 180,E1 -13378.942,E2 -13378.942} C_VEL
LIN {X 0,Y 359.971,Z 609.058,A -85,B 0,C 180,E1 -13381.746,E2 -13381.746} C_VEL
LIN {X 0,Y 360.305,Z 611.949,A -85,B 0,C 180,E1 -13382.403,E2 -13382.403} C_VEL
LIN {X 0,Y 358.368,Z 629.255,A -85,B 0,C 180,E1 -13385.988,E2 -13385.988} C_VEL
LIN {X 0,Y 357.973,Z 633.55,A -85,B 0,C 180,E1 -13386.828,E2 -13386.828} C_VEL
LIN {X 0,Y 361.224,Z 653.183,A -85,B 0,C 180,E1 -13387.554,E2 -13387.554} C_VEL
LIN {X 0,Y 364.072,Z 678.339,A -85,B 0,C 180,E1 -13388.355,E2 -13388.355} C_VEL
LIN {X 0,Y 362.548,Z 744.922,A -85,B 0,C 180,E1 -13389.838,E2 -13389.838} C_VEL
LIN {X 0,Y 361.708,Z 758.21,A -85,B 0,C 180,E1 -13390.344,E2 -13390.344} C_VEL
LIN {X 0,Y 360.681,Z 770.485,A -85,B 0,C 180,E1 -13391.025,E2 -13391.025} C_VEL
LIN {X 0,Y 359.454,Z 782.427,A -85,B 0,C 180,E1 -13391.918,E2 -13391.918} C_VEL
LIN {X 0,Y 358.199,Z 793.978,A -85,B 0,C 180,E1 -13393.032,E2 -13393.032} C_VEL
LIN {X 0,Y 357.013,Z 804.461,A -85,B 0,C 180,E1 -13394.296,E2 -13394.296} C_VEL
LIN {X 0,Y 356.077,Z 813.925,A -85,B 0,C 180,E1 -13395.717,E2 -13395.717} C_VEL
LIN {X 0,Y 355.12,Z 821.756,A -85,B 0,C 180,E1 -13397.136,E2 -13397.136} C_VEL
LIN {X 0,Y 354.294,Z 829.476,A -85,B 0,C 180,E1 -13398.849,E2 -13398.849} C_VEL
LIN {X 0,Y 353.911,Z 834.772,A -85,B 0,C 180,E1 -13400.283,E2 -13400.283} C_VEL
LIN {X 0,Y 353.625,Z 839.938,A -85,B 0,C 180,E1 -13402.003,E2 -13402.003} C_VEL
LIN {X 0,Y 353.506,Z 844.003,A -85,B 0,C 180,E1 -13403.745,E2 -13403.745} C_VEL
LIN {X 0,Y 353.482,Z 846.926,A -85,B 0,C 180,E1 -13405.439,E2 -13405.439} C_VEL
LIN {X 0,Y 353.54,Z 848.353,A -85,B 0,C 180,E1 -13406.581,E2 -13406.581} C_VEL
LIN {X 0,Y 353.663,Z 849.374,A -85,B 0,C 180,E1 -13407.722,E2 -13407.722} C_VEL
LIN {X 0,Y 353.697,Z 849.947,A -85,B 0,C 180,E1 -13408.861,E2 -13408.861} C_VEL
LIN {X 0,Y 353.726,Z 850.085,A -85,B 0,C 180,E1 -13410,E2 -13410} C_VEL
LIN {X 0,Y 353.744,Z 849.818,A -85,B 0,C 180,E1 -13411.138,E2 -13411.138} C_VEL
LIN {X 0,Y 353.685,Z 849.138,A -85,B 0,C 180,E1 -13412.278,E2 -13412.278} C_VEL
LIN {X 0,Y 353.595,Z 848,A -85,B 0,C 180,E1 -13413.418,E2 -13413.418} C_VEL
LIN {X 0,Y 353.523,Z 845.484,A -85,B 0,C 180,E1 -13415.132,E2 -13415.132} C_VEL
LIN {X 0,Y 353.523,Z 840.665,A -85,B 0,C 180,E1 -13417.424,E2 -13417.424} C_VEL
LIN {X 0,Y 353.757,Z 836.165,A -85,B 0,C 180,E1 -13419.145,E2 -13419.145} C_VEL
LIN {X 0,Y 354.177,Z 830.472,A -85,B 0,C 180,E1 -13420.866,E2 -13420.866} C_VEL
LIN {X 0,Y 354.994,Z 823.379,A -85,B 0,C 180,E1 -13422.578,E2 -13422.578} C_VEL
LIN {X 0,Y 356.018,Z 814.694,A -85,B 0,C 180,E1 -13424.257,E2 -13424.257} C_VEL
LIN {X 0,Y 356.998,Z 805.489,A -85,B 0,C 180,E1 -13425.704,E2 -13425.704} C_VEL
LIN {X 0,Y 358.27,Z 795.535,A -85,B 0,C 180,E1 -13426.965,E2 -13426.965} C_VEL
LIN {X 0,Y 359.649,Z 784.484,A -85,B 0,C 180,E1 -13428.072,E2 -13428.072} C_VEL
LIN {X 0,Y 360.842,Z 772.124,A -85,B 0,C 180,E1 -13429.04,E2 -13429.04} C_VEL
LIN {X 0,Y 362.001,Z 759.532,A -85,B 0,C 180,E1 -13429.75,E2 -13429.75} C_VEL
LIN {X 0,Y 362.831,Z 746.21,A -85,B 0,C 180,E1 -13430.257,E2 -13430.257} C_VEL
LIN {X 0,Y 363.456,Z 717.418,A -85,B 0,C 180,E1 -13430.875,E2 -13430.875} C_VEL
LIN {X 0,Y 364.096,Z 674.246,A -85,B 0,C 180,E1 -13431.755,E2 -13431.755} C_VEL
LIN {X 0,Y 360.758,Z 645.154,A -85,B 0,C 180,E1 -13432.632,E2 -13432.632} C_VEL
LIN {X 0,Y 358.53,Z 629.722,A -85,B 0,C 180,E1 -13433.158,E2 -13433.158} C_VEL
LIN {X 0,Y 360.301,Z 611.512,A -85,B 0,C 180,E1 -13436.331,E2 -13436.331} C_VEL
LIN {X 0,Y 359.104,Z 604.375,A -85,B 0,C 180,E1 -13437.697,E2 -13437.697} C_VEL
LIN {X 0,Y 355.258,Z 588.236,A -85,B 0,C 180,E1 -13440.953,E2 -13440.953} C_VEL
LIN {X 0,Y 354.803,Z 586.291,A -85,B 0,C 180,E1 -13441.381,E2 -13441.381} C_VEL
LIN {X 0,Y 354.811,Z 586.287,A -85,B 0,C 180,E1 -13445.058,E2 -13445.058} C_VEL
LIN {X 0,Y 354.809,Z 586.285,A -85,B 0,C 180,E1 -13447.881,E2 -13447.881} C_VEL
LIN {X 0,Y 354.813,Z 586.284,A -85,B 0,C 180,E1 -13451.176,E2 -13451.176} C_VEL
LIN {X 0,Y 354.827,Z 586.283,A -85,B 0,C 180,E1 -13454.517,E2 -13454.517} C_VEL
LIN {X 0,Y 354.834,Z 586.284,A -85,B 0,C 180,E1 -13457.668,E2 -13457.668} C_VEL
LIN {X 0,Y 354.833,Z 586.277,A -85,B 0,C 180,E1 -13460.668,E2 -13460.668} C_VEL
LIN {X 0,Y 354.817,Z 586.279,A -85,B 0,C 180,E1 -13464.3,E2 -13464.3} C_VEL
LIN {X 0,Y 354.792,Z 586.288,A -85,B 0,C 180,E1 -13467.667,E2 -13467.667} C_VEL
LIN {X 0,Y 354.863,Z 586.267,A -85,B 0,C 180,E1 -13470.621,E2 -13470.621} C_VEL
LIN {X 0,Y 354.893,Z 586.279,A -85,B 0,C 180,E1 -13474.172,E2 -13474.172} C_VEL
LIN {X 0,Y 354.827,Z 586.268,A -85,B 0,C 180,E1 -13477.893,E2 -13477.893} C_VEL
LIN {X 0,Y 354.915,Z 586.273,A -85,B 0,C 180,E1 -13481.891,E2 -13481.891} C_VEL
LIN {X 0,Y 354.935,Z 586.265,A -85,B 0,C 180,E1 -13485.981,E2 -13485.981} C_VEL
LIN {X 0,Y 354.97,Z 586.259,A -85,B 0,C 180,E1 -13489.736,E2 -13489.736} C_VEL
LIN {X 0,Y 355.121,Z 586.246,A -85,B 0,C 180,E1 -13493.18,E2 -13493.18} C_VEL
LIN {X 0,Y 355.238,Z 586.219,A -85,B 0,C 180,E1 -13497.732,E2 -13497.732} C_VEL
LIN {X 0,Y 355.39,Z 586.205,A -85,B 0,C 180,E1 -13500,E2 -13500} C_VEL
LIN {X 0,Y 355.238,Z 586.234,A -85,B 0,C 180,E1 -13502.268,E2 -13502.268} C_VEL
LIN {X 0,Y 355.119,Z 586.236,A -85,B 0,C 180,E1 -13506.82,E2 -13506.82} C_VEL
LIN {X 0,Y 354.97,Z 586.267,A -85,B 0,C 180,E1 -13510.264,E2 -13510.264} C_VEL
LIN {X 0,Y 354.935,Z 586.265,A -85,B 0,C 180,E1 -13514.019,E2 -13514.019} C_VEL
LIN {X 0,Y 354.915,Z 586.265,A -85,B 0,C 180,E1 -13518.109,E2 -13518.109} C_VEL
LIN {X 0,Y 354.822,Z 586.285,A -85,B 0,C 180,E1 -13522.107,E2 -13522.107} C_VEL
LIN {X 0,Y 354.892,Z 586.273,A -85,B 0,C 180,E1 -13525.828,E2 -13525.828} C_VEL
LIN {X 0,Y 354.848,Z 586.272,A -85,B 0,C 180,E1 -13529.679,E2 -13529.679} C_VEL
LIN {X 0,Y 354.825,Z 586.278,A -85,B 0,C 180,E1 -13533.683,E2 -13533.683} C_VEL
LIN {X 0,Y 354.794,Z 586.289,A -85,B 0,C 180,E1 -13536.46,E2 -13536.46} C_VEL
LIN {X 0,Y 354.819,Z 586.285,A -85,B 0,C 180,E1 -13539.424,E2 -13539.424} C_VEL
LIN {X 0,Y 354.8,Z 586.265,A -85,B 0,C 180,E1 -13542.871,E2 -13542.871} C_VEL
LIN {X 0,Y 354.778,Z 586.288,A -85,B 0,C 180,E1 -13546.107,E2 -13546.107} C_VEL
LIN {X 0,Y 354.785,Z 586.285,A -85,B 0,C 180,E1 -13549.18,E2 -13549.18} C_VEL
LIN {X 0,Y 354.806,Z 586.277,A -85,B 0,C 180,E1 -13552.403,E2 -13552.403} C_VEL
LIN {X 0,Y 354.827,Z 586.285,A -85,B 0,C 180,E1 -13554.529,E2 -13554.529} C_VEL
LIN {X 0,Y 355.971,Z 589.333,A -85,B 0,C 180,E1 -13554.72,E2 -13554.72} C_VEL
LIN {X 0,Y 364.58,Z 607.207,A -85,B 0,C 180,E1 -13555.804,E2 -13555.804} C_VEL
LIN {X 0,Y 365.825,Z 610.135,A -85,B 0,C 180,E1 -13555.962,E2 -13555.962} C_VEL
LIN {X 0,Y 364.367,Z 684.568,A -85,B 0,C 180,E1 -13557.466,E2 -13557.466} C_VEL
LIN {X 0,Y 363.993,Z 697.529,A -85,B 0,C 180,E1 -13557.926,E2 -13557.926} C_VEL
LIN {X 0,Y 363.383,Z 710.127,A -85,B 0,C 180,E1 -13558.603,E2 -13558.603} C_VEL
LIN {X 0,Y 362.487,Z 721.265,A -85,B 0,C 180,E1 -13559.407,E2 -13559.407} C_VEL
LIN {X 0,Y 361.429,Z 732.315,A -85,B 0,C 180,E1 -13560.435,E2 -13560.435} C_VEL
LIN {X 0,Y 360.227,Z 742.936,A -85,B 0,C 180,E1 -13561.678,E2 -13561.678} C_VEL
LIN {X 0,Y 359.126,Z 751.607,A -85,B 0,C 180,E1 -13562.936,E2 -13562.936} C_VEL
LIN {X 0,Y 357.896,Z 760.832,A -85,B 0,C 180,E1 -13564.596,E2 -13564.596} C_VEL
LIN {X 0,Y 356.831,Z 767.983,A -85,B 0,C 180,E1 -13566.187,E2 -13566.187} C_VEL
LIN {X 0,Y 355.89,Z 774.36,A -85,B 0,C 180,E1 -13567.964,E2 -13567.964} C_VEL
LIN {X 0,Y 355.137,Z 779.33,A -85,B 0,C 180,E1 -13569.738,E2 -13569.738} C_VEL
LIN {X 0,Y 354.594,Z 783.096,A -85,B 0,C 180,E1 -13571.512,E2 -13571.512} C_VEL
LIN {X 0,Y 354.311,Z 785.007,A -85,B 0,C 180,E1 -13572.691,E2 -13572.691} C_VEL
LIN {X 0,Y 354.019,Z 786.483,A -85,B 0,C 180,E1 -13573.864,E2 -13573.864} C_VEL
LIN {X 0,Y 353.837,Z 787.485,A -85,B 0,C 180,E1 -13575.037,E2 -13575.037} C_VEL
LIN {X 0,Y 353.715,Z 788.235,A -85,B 0,C 180,E1 -13576.803,E2 -13576.803} C_VEL
LIN {X 0,Y 353.66,Z 788.065,A -85,B 0,C 180,E1 -13578.538,E2 -13578.538} C_VEL
LIN {X 0,Y 353.715,Z 786.422,A -85,B 0,C 180,E1 -13580.854,E2 -13580.854} C_VEL
LIN {X 0,Y 353.874,Z 784.975,A -85,B 0,C 180,E1 -13582.009,E2 -13582.009} C_VEL
LIN {X 0,Y 354.144,Z 782.001,A -85,B 0,C 180,E1 -13583.734,E2 -13583.734} C_VEL
LIN {X 0,Y 354.472,Z 777.994,A -85,B 0,C 180,E1 -13585.451,E2 -13585.451} C_VEL
LIN {X 0,Y 354.903,Z 772.841,A -85,B 0,C 180,E1 -13587.162,E2 -13587.162} C_VEL
LIN {X 0,Y 355.581,Z 766.361,A -85,B 0,C 180,E1 -13588.868,E2 -13588.868} C_VEL
LIN {X 0,Y 356.375,Z 758.335,A -85,B 0,C 180,E1 -13590.565,E2 -13590.565} C_VEL
LIN {X 0,Y 357.244,Z 750.071,A -85,B 0,C 180,E1 -13591.973,E2 -13591.973} C_VEL
LIN {X 0,Y 358.136,Z 739.951,A -85,B 0,C 180,E1 -13593.375,E2 -13593.375} C_VEL
LIN {X 0,Y 358.983,Z 729.973,A -85,B 0,C 180,E1 -13594.491,E2 -13594.491} C_VEL
LIN {X 0,Y 359.849,Z 719.082,A -85,B 0,C 180,E1 -13595.463,E2 -13595.463} C_VEL
LIN {X 0,Y 360.52,Z 706.91,A -85,B 0,C 180,E1 -13596.295,E2 -13596.295} C_VEL
LIN {X 0,Y 361.036,Z 693.527,A -85,B 0,C 180,E1 -13596.953,E2 -13596.953} C_VEL
LIN {X 0,Y 361.357,Z 681.189,A -85,B 0,C 180,E1 -13597.333,E2 -13597.333} C_VEL
LIN {X 0,Y 362.402,Z 606.102,A -85,B 0,C 180,E1 -13598.822,E2 -13598.822} C_VEL
LIN {X 0,Y 355.058,Z 586.643,A -85,B 0,C 180,E1 -13599.614,E2 -13599.614} C_VEL
LIN {X 0,Y 355.016,Z 586.263,A -85,B 0,C 180,E1 -13599.687,E2 -13599.687} C_VEL
LIN {X 0,Y 354.943,Z 586.27,A -85,B 0,C 180,E1 -13603.613,E2 -13603.613} C_VEL
LIN {X 0,Y 354.331,Z 586.352,A -85,B 0,C 180,E1 -13604.559,E2 -13604.559} C_VEL
LIN {X 0,Y 351.496,Z 586.709,A -85,B 0,C 180,E1 -13606.098,E2 -13606.098} C_VEL
LIN {X 0,Y 349.044,Z 587.012,A -85,B 0,C 180,E1 -13607.343,E2 -13607.343} C_VEL
LIN {X 0,Y 347.966,Z 587.143,A -85,B 0,C 180,E1 -13608.307,E2 -13608.307} C_VEL
LIN {X 0,Y 347.867,Z 587.153,A -85,B 0,C 180,E1 -13608.634,E2 -13608.634} C_VEL
LIN {X 0,Y 347.762,Z 587.165,A -85,B 0,C 180,E1 -13612.58,E2 -13612.58} C_VEL
LIN {X 0,Y 347.821,Z 587.158,A -85,B 0,C 180,E1 -13613.638,E2 -13613.638} C_VEL
LIN {X 0,Y 350.227,Z 593.66,A -85,B 0,C 180,E1 -13613.949,E2 -13613.949} C_VEL
LIN {X 0,Y 356.379,Z 609.16,A -85,B 0,C 180,E1 -13614.667,E2 -13614.667} C_VEL
LIN {X 0,Y 354.801,Z 684.757,A -85,B 0,C 180,E1 -13616.324,E2 -13616.324} C_VEL
LIN {X 0,Y 354.362,Z 697.729,A -85,B 0,C 180,E1 -13616.813,E2 -13616.813} C_VEL
LIN {X 0,Y 353.844,Z 710.057,A -85,B 0,C 180,E1 -13617.502,E2 -13617.502} C_VEL
LIN {X 0,Y 353.038,Z 721.85,A -85,B 0,C 180,E1 -13618.377,E2 -13618.377} C_VEL
LIN {X 0,Y 352.184,Z 733.121,A -85,B 0,C 180,E1 -13619.466,E2 -13619.466} C_VEL
LIN {X 0,Y 351.222,Z 743.605,A -85,B 0,C 180,E1 -13620.732,E2 -13620.732} C_VEL
LIN {X 0,Y 350.268,Z 752.952,A -85,B 0,C 180,E1 -13622.12,E2 -13622.12} C_VEL
LIN {X 0,Y 349.432,Z 760.988,A -85,B 0,C 180,E1 -13623.579,E2 -13623.579} C_VEL
LIN {X 0,Y 348.678,Z 767.719,A -85,B 0,C 180,E1 -13625.059,E2 -13625.059} C_VEL
LIN {X 0,Y 348.07,Z 773.776,A -85,B 0,C 180,E1 -13626.688,E2 -13626.688} C_VEL
LIN {X 0,Y 347.441,Z 779.969,A -85,B 0,C 180,E1 -13628.833,E2 -13628.833} C_VEL
LIN {X 0,Y 347.067,Z 783.397,A -85,B 0,C 180,E1 -13630.389,E2 -13630.389} C_VEL
LIN {X 0,Y 346.796,Z 786.049,A -85,B 0,C 180,E1 -13631.97,E2 -13631.97} C_VEL
LIN {X 0,Y 346.597,Z 787.93,A -85,B 0,C 180,E1 -13633.583,E2 -13633.583} C_VEL
LIN {X 0,Y 346.508,Z 789.006,A -85,B 0,C 180,E1 -13635.224,E2 -13635.224} C_VEL
LIN {X 0,Y 346.569,Z 789.288,A -85,B 0,C 180,E1 -13636.888,E2 -13636.888} C_VEL
LIN {X 0,Y 346.677,Z 788.737,A -85,B 0,C 180,E1 -13638.596,E2 -13638.596} C_VEL
LIN {X 0,Y 346.969,Z 787.284,A -85,B 0,C 180,E1 -13640.326,E2 -13640.326} C_VEL
LIN {X 0,Y 347.396,Z 784.84,A -85,B 0,C 180,E1 -13642.089,E2 -13642.089} C_VEL
LIN {X 0,Y 347.951,Z 780.679,A -85,B 0,C 180,E1 -13644.144,E2 -13644.144} C_VEL
LIN {X 0,Y 348.708,Z 775.332,A -85,B 0,C 180,E1 -13646.088,E2 -13646.088} C_VEL
LIN {X 0,Y 349.508,Z 769.953,A -85,B 0,C 180,E1 -13647.621,E2 -13647.621} C_VEL
LIN {X 0,Y 350.577,Z 762.426,A -85,B 0,C 180,E1 -13649.358,E2 -13649.358} C_VEL
LIN {X 0,Y 351.798,Z 753.331,A -85,B 0,C 180,E1 -13651.023,E2 -13651.023} C_VEL
LIN {X 0,Y 352.984,Z 743.843,A -85,B 0,C 180,E1 -13652.425,E2 -13652.425} C_VEL
LIN {X 0,Y 354.036,Z 733.886,A -85,B 0,C 180,E1 -13653.619,E2 -13653.619} C_VEL
LIN {X 0,Y 355.1,Z 722.128,A -85,B 0,C 180,E1 -13654.73,E2 -13654.73} C_VEL
LIN {X 0,Y 356.005,Z 710.335,A -85,B 0,C 180,E1 -13655.585,E2 -13655.585} C_VEL
LIN {X 0,Y 356.612,Z 697.198,A -85,B 0,C 180,E1 -13656.287,E2 -13656.287} C_VEL
LIN {X 0,Y 356.975,Z 685.57,A -85,B 0,C 180,E1 -13656.697,E2 -13656.697} C_VEL
LIN {X 0,Y 358.882,Z 611.322,A -85,B 0,C 180,E1 -13658.372,E2 -13658.372} C_VEL
LIN {X 0,Y 351.855,Z 595.988,A -85,B 0,C 180,E1 -13659.342,E2 -13659.342} C_VEL
LIN {X 0,Y 347.941,Z 587.957,A -85,B 0,C 180,E1 -13659.896,E2 -13659.896} C_VEL
LIN {X 0,Y 347.805,Z 587.162,A -85,B 0,C 180,E1 -13659.986,E2 -13659.986} C_VEL
LIN {X 0,Y 347.859,Z 587.156,A -85,B 0,C 180,E1 -13662.359,E2 -13662.359} C_VEL
LIN {X 0,Y 347.89,Z 587.153,A -85,B 0,C 180,E1 -13665.97,E2 -13665.97} C_VEL
LIN {X 0,Y 347.925,Z 587.146,A -85,B 0,C 180,E1 -13669.525,E2 -13669.525} C_VEL
LIN {X 0,Y 348.066,Z 587.129,A -85,B 0,C 180,E1 -13671.875,E2 -13671.875} C_VEL
LIN {X 0,Y 348.064,Z 587.131,A -85,B 0,C 180,E1 -13674.206,E2 -13674.206} C_VEL
LIN {X 0,Y 348.201,Z 587.107,A -85,B 0,C 180,E1 -13677.686,E2 -13677.686} C_VEL
LIN {X 0,Y 348.36,Z 587.091,A -85,B 0,C 180,E1 -13680,E2 -13680} C_VEL
LIN {X 0,Y 348.2,Z 587.114,A -85,B 0,C 180,E1 -13682.314,E2 -13682.314} C_VEL
LIN {X 0,Y 348.09,Z 587.118,A -85,B 0,C 180,E1 -13686.958,E2 -13686.958} C_VEL
LIN {X 0,Y 347.925,Z 587.137,A -85,B 0,C 180,E1 -13690.475,E2 -13690.475} C_VEL
LIN {X 0,Y 347.891,Z 587.139,A -85,B 0,C 180,E1 -13694.15,E2 -13694.15} C_VEL
LIN {X 0,Y 347.884,Z 587.145,A -85,B 0,C 180,E1 -13698.291,E2 -13698.291} C_VEL
LIN {X 0,Y 347.781,Z 587.159,A -85,B 0,C 180,E1 -13701.635,E2 -13701.635} C_VEL
LIN {X 0,Y 347.806,Z 587.16,A -85,B 0,C 180,E1 -13705.109,E2 -13705.109} C_VEL
LIN {X 0,Y 347.806,Z 587.153,A -85,B 0,C 180,E1 -13707.694,E2 -13707.694} C_VEL
LIN {X 0,Y 347.759,Z 587.163,A -85,B 0,C 180,E1 -13710.347,E2 -13710.347} C_VEL
LIN {X 0,Y 347.739,Z 587.167,A -85,B 0,C 180,E1 -13714.465,E2 -13714.465} C_VEL
LIN {X 0,Y 347.772,Z 587.165,A -85,B 0,C 180,E1 -13717.99,E2 -13717.99} C_VEL
LIN {X 0,Y 347.78,Z 587.16,A -85,B 0,C 180,E1 -13721.61,E2 -13721.61} C_VEL
LIN {X 0,Y 347.794,Z 587.164,A -85,B 0,C 180,E1 -13725.012,E2 -13725.012} C_VEL
LIN {X 0,Y 347.765,Z 587.169,A -85,B 0,C 180,E1 -13728.395,E2 -13728.395} C_VEL
LIN {X 0,Y 347.774,Z 587.166,A -85,B 0,C 180,E1 -13732.012,E2 -13732.012} C_VEL
